// TIA Portal V20 export
// export: Created 2025-12-01T14:56:29.3787725Z, ExportSetting None, DisplayName Totally Integrated Automation Portal, DisplayVersion V20 Update 3, DisplayName TIA Portal Openness, DisplayVersion V20 Update 3, DisplayName TIA Portal Version Control Interface, DisplayVersion V20 Update 3, DisplayName STEP 7 Professional, DisplayVersion V20 Update 3, DisplayName STEP 7 Safety, DisplayVersion V20 Update 2, DisplayName WinCC Basic/Comfort/Advanced, DisplayVersion V20 Update 3, DisplayName WinCC Professional, DisplayVersion V20 Update 3, DisplayName WinCC Unified, DisplayVersion V20 Update 3
FUNCTION_BLOCK "FB430_CRTL_Emp_TP_E1_S23"   // FB430, LAD
{ S7_Optimized_Access := 'FALSE' }
AUTHOR : ROUTER
NAME : 20180827
VERSION : 3.1
// ////////////////////////////////////////////////////////////////
// /  Modificada  24/08/15          NIEVES RODRIGUEZ              /
// /                               /
// ////////////////////////////////////////////////////////////////
// stored: AutoNumber false, SetENOAutomatically false
   VAR_INPUT
      Mesa : UInt;   // Número de mesa
      En_Tension : Bool;
      pHsMx_E1 : Bool;   // pHs de ausencia de la Mesa por E1
      pHsMx_S3 : Bool;   // pHs de ausencia de la Mesa por S3
      Termico_Tx : Bool;   // Proteccion del Tx en E1E3
      Avance_Tx : Bool;   // Avance del Tx
      TP1_Up : Bool;   // TP1 Arriba. E1 >> S3. si no hay tope poner ON
      TP1_Down : Bool;   // TP1 Abajo. E1 >> S3. si no hay tope poner ON
      Simul_Mx : Bool;   // Permiso de Simultaneo en la Entrada E1
      IN_Empuj_recogido : Bool;   // Empujador recogido
      IN_Empuj_Extendido : Bool;   // Empujador extendido
      Mx_Bloq_Activo_S2 : Bool;   // Bloqueo Activo de la Mesa
      AVTF_MAnt_Mx : Bool;   // E1 >> Mesa Anterior AVTF
      PTF_Sal_M3 : Bool;   // S3 >> Mesa Siguiente PTF
      NXT_Avance_S3 : Bool;   // S3 >> Mesa Siguiente avanzando
      PTF_Sal_M2 : Bool;   // Desactiva si Transferencia controlada
      NXT_Avance_S2 : Bool;   // S2 >> Mesa Siguiente avanzando
      F_EnvMens_Mx : Bool;   // Fin de Envio de Mensaje
      Num_Cruce : UInt;   // Número de cruce.
      DB_FIFO_Cruce : UInt := 213;   // DB de la FIFO de ordenes del cruce
      Lng_FIFO_Cruce : UInt := 1;   // Longitut de la FIFO de ordenes del cruce
      ValorOrden_S2 : Word := 16#81;   // Con que orden entra por S2
      MesaS2 : UInt;   // Número de mesa por S2
      MesaS3 : UInt;   // Número de mesa por S3
      V_Paro : UDInt := 4000;   // tiempo que avanza el transportador sin aviso hasta que se para (ms)
      V_CNT_ApHsMx_E1 : UDInt := 500;   // Valor de Ausencia por E1 en ms
      V_CNT_ApHsMx_S3 : UDInt := 500;   // Valor de Ausencia por S3 en ms
      V_Vaciado : UDInt := 3000;   // Valor de vaciado en ms
      V_Gap : UDInt := 200;   // espacio que se deja antes de iniciar un simultaneo en ms
      V_TOut_empujador : UDInt := 2000;   // TimeOut del empujador en ms
      V_TOut_TP : UDInt := 2000;   // TimeOut de Tope en ms
   END_VAR
   VAR_OUTPUT
      P_EnvMens_PMx : Bool;   // Permiso de Enviar Mensaje de Presencia
      Etiqueta_Jdt : UDInt;   // Etiqueta que ha sido leida
      Orden_Ejecutada_Jdt : UInt;   // Orden que se ha ejecutado
      PTF_MAnt_Mx : Bool;   // E1 >> Mesa Anterior PTF
      AVTF_Sal_M3 : Bool;   // S3 >> Mesa Siguiente AVTF
      NXT_Descarga_Act_S3 : Bool;   // S3 >> Mesa Siguiente Descarga activa
      AVTF_Sal_M2 : Bool;   // S2 >> Mesa Siguiente AVTF
      NXT_Descarga_Act_S2 : Bool;   // S2 >> Mesa Siguiente Descarga activa
   END_VAR
   VAR
      T1_ET00 : Bool;
      T1_ET01 : Bool;
      T1_ET02 : Bool;
      T1_ET03 : Bool;
      T1_ET10 : Bool;
      T1_ET11 : Bool;
      T1_ET50 : Bool;
      T1_ET60 : Bool;
      T1_ET61 : Bool;
      T1_ET110 : Bool;
      T1_ET111 : Bool;
      T1_ET112 : Bool;
      FIFO_OK : Bool;
      TRANS_OK : Bool;
      O_Bloqueo : Bool;
      FN_ET02 : Bool;
      FP_ET50 : Bool;
      FP_Bajar_TP : Bool;
      TOUT_empujador : Bool;
      ok_vaciado : Bool;
      maux_fp_disparo : Bool;
      maux_fn_s3 : Bool;
      maux_fn_e1 : Bool;
      mem_fn_e1 : Bool;
      mem_fn_s3 : Bool;
      TmpSIMUL : UDInt;
      Tmp_Ausencia : UDInt;
      Tmp_Vaciado : UDInt;
      tmp_tout_empujador : UDInt;
      Tmp_tout_tope : UDInt;
      tmp_ausencia_S3 : UDInt;
      TMP_Paro : UDInt;
      TMP_En_tension : UDInt;
      Datos_Scanner { S7_SetPoint := 'True'} : "ROUT_Orden_Fifo_Scanner";
   END_VAR
   VAR_TEMP
      EstadoZona : "EstadoZona";   // Estado de Zona de la Mesa
      EstadoVI : "EstadosMesa";   // Estado del Vehiculo Inteliguente de la Mesa
      ConfigFB : "UDT_ConfigFB";   // Configuracion de la FB de la Mesa
      OK_tension : Bool;
      MA_SubirTP : Bool;
      O_Sal_S3 : Bool;
      O_Sal_S2 : Bool;
      O_Vaciar : Bool;
      Moti_ERRO : Bool;
      Moti_NENC : Bool;
      Moti_NORM : Bool;
      Moti_INIC : Bool;
      OK_SIMUL_S3 : Bool;
      ok_ausencia_S3 : Bool;
      tout_tope : Bool;
      ok_ausencia_E1 : Bool;
      tiempo_paro_ok : Bool;
      INT_ORDEN : UInt;
      I_Ord_Filtrada : UInt;
      I_V_Ord_Entrar : UInt;
      Prox_Orden : UInt;
      Prox_Etiqueta : DInt;
      Aux_W_Orden : Word;
      Aux_W_Moti : Word;
   END_VAR
   VAR_TEMP   // added for the SCL form of the ladder/FBD networks
      _w1 : Bool;
      _w2 : Bool;
      _w3 : Bool;
      _w4 : Bool;
      _w5 : Bool;
      _w6 : Bool;
   END_VAR
BEGIN

REGION Network 1: INICIALIZAR - Recoger las Variables de Estado de la Mesa
   // Se recoge - Estado_CBx
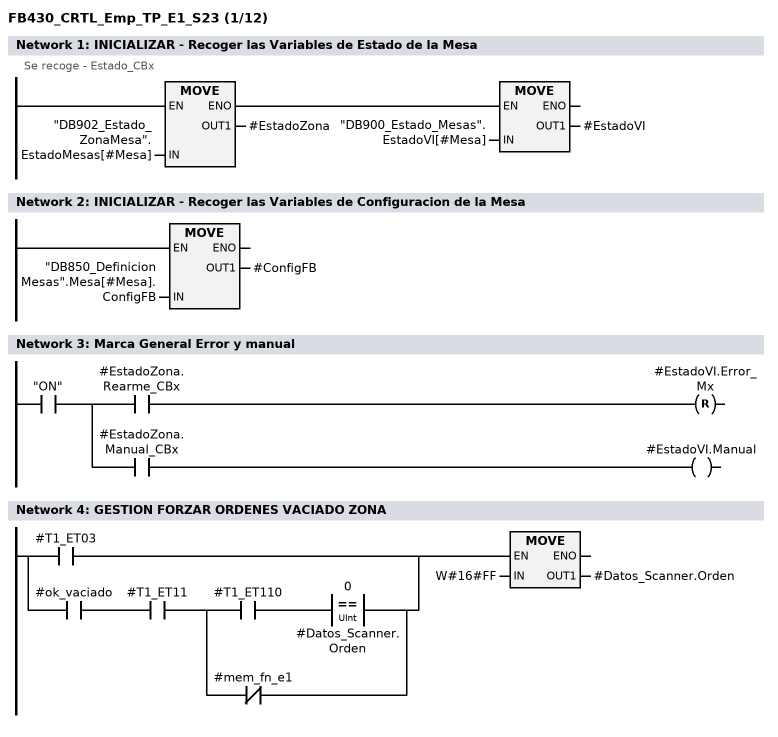
   RUNG wire#powerrail
      Move(in := "DB902_Estado_ZonaMesa".EstadoMesas[#Mesa], out1 => #EstadoZona)
      Move(in := "DB900_Estado_Mesas".EstadoVI[#Mesa], out1 => #EstadoVI)
   END_RUNG
   // the same network as SCL:
   #EstadoZona := "DB902_Estado_ZonaMesa".EstadoMesas[#Mesa];
   #EstadoVI := "DB900_Estado_Mesas".EstadoVI[#Mesa];
END_REGION

REGION Network 2: INICIALIZAR - Recoger las Variables de Configuracion de la Mesa
   RUNG wire#powerrail
      Move(in := "DB850_DefinicionMesas".Mesa[#Mesa].ConfigFB, out1 => #ConfigFB)
   END_RUNG
   // the same network as SCL:
   #ConfigFB := "DB850_DefinicionMesas".Mesa[#Mesa].ConfigFB;
END_REGION

REGION Network 3: Marca General Error y manual
   RUNG wire#powerrail
      Contact( "ON" )
      wire#w1
      Contact( #EstadoZona.Rearme_CBx )
      R_Coil( #EstadoVI.Error_Mx )
   END_RUNG
   RUNG wire#w1
      Contact( #EstadoZona.Manual_CBx )
      Coil( #EstadoVI.Manual )
   END_RUNG
   // the same network as SCL:
   IF "ON" AND #EstadoZona.Rearme_CBx THEN #EstadoVI.Error_Mx := FALSE; END_IF;
   #EstadoVI.Manual := "ON" AND #EstadoZona.Manual_CBx;
END_REGION

REGION Network 4: GESTION FORZAR ORDENES VACIADO ZONA
   RUNG wire#powerrail
      Contact( #T1_ET03 )
      wire#w1
      { S7_GenerateENO := "TRUE" } Move(in := W#16#FF, out1 => #Datos_Scanner.Orden)
   END_RUNG
   RUNG wire#powerrail
      Contact( #ok_vaciado )
      Contact( #T1_ET11 )
      wire#w2
      Contact( #T1_ET110 )
      { S7_Templates := "SrcType := UInt" } EQ_Contact(in1 := 0, in2 := #Datos_Scanner.Orden)
   END_RUNG wire#w1
   RUNG wire#w2
      I_Contact( #mem_fn_e1 )
   END_RUNG wire#w1
   // the same network as SCL:
   IF #T1_ET03 OR (#ok_vaciado AND #T1_ET11 AND ((#T1_ET110 AND (0 = #Datos_Scanner.Orden)) OR NOT #mem_fn_e1)) THEN
       #Datos_Scanner.Orden := W#16#FF;
   END_IF;
END_REGION

REGION Network 5: Extraccion de orden
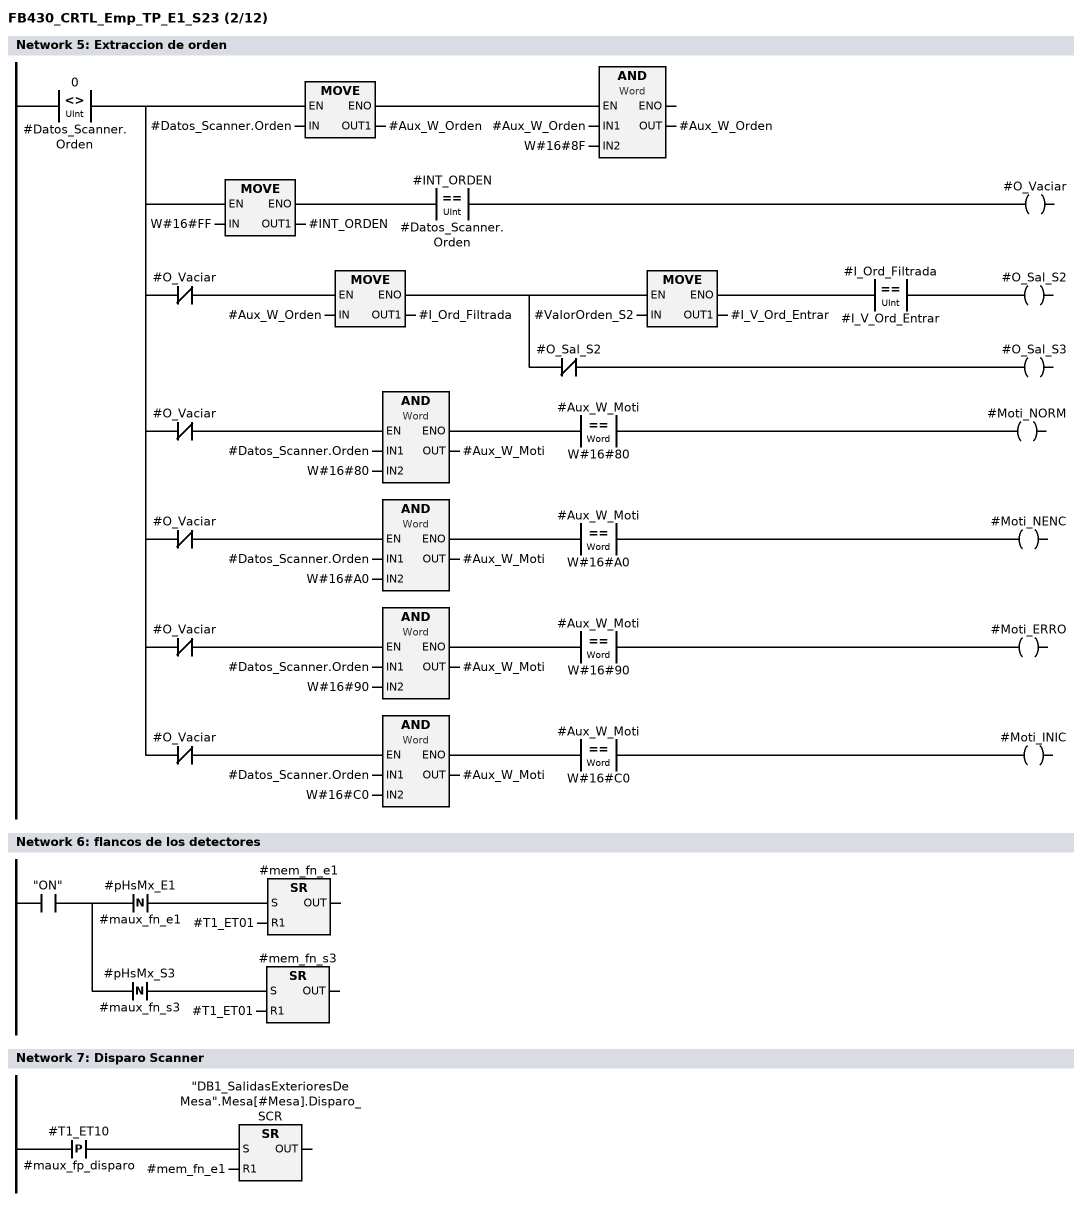
   RUNG wire#powerrail
      { S7_Templates := "SrcType := UInt" } NE_Contact(in1 := 0, in2 := #Datos_Scanner.Orden)
      wire#w1
      { S7_GenerateENO := "TRUE" } Move(in := #Datos_Scanner.Orden, out1 => #Aux_W_Orden)
      { S7_Templates := "SrcType := Word"; S7_GenerateENO := "TRUE" } And(in1 := #Aux_W_Orden, in2 := W#16#8F, out => #Aux_W_Orden)
   END_RUNG
   RUNG wire#w1
      { S7_GenerateENO := "TRUE" } Move(in := W#16#FF, out1 => #INT_ORDEN)
      { S7_Templates := "SrcType := UInt" } EQ_Contact(in1 := #INT_ORDEN, in2 := #Datos_Scanner.Orden)
      Coil( #O_Vaciar )
   END_RUNG
   RUNG wire#w1
      I_Contact( #O_Vaciar )
      { S7_GenerateENO := "TRUE" } Move(in := #Aux_W_Orden, out1 => #I_Ord_Filtrada)
      wire#w2
      { S7_GenerateENO := "TRUE" } Move(in := #ValorOrden_S2, out1 => #I_V_Ord_Entrar)
      { S7_Templates := "SrcType := UInt" } EQ_Contact(in1 := #I_Ord_Filtrada, in2 := #I_V_Ord_Entrar)
      Coil( #O_Sal_S2 )
   END_RUNG
   RUNG wire#w2
      I_Contact( #O_Sal_S2 )
      Coil( #O_Sal_S3 )
   END_RUNG
   RUNG wire#w1
      I_Contact( #O_Vaciar )
      { S7_Templates := "SrcType := Word"; S7_GenerateENO := "TRUE" } And(in1 := #Datos_Scanner.Orden, in2 := W#16#80, out => #Aux_W_Moti)
      { S7_Templates := "SrcType := Word" } EQ_Contact(in1 := #Aux_W_Moti, in2 := W#16#80)
      Coil( #Moti_NORM )
   END_RUNG
   RUNG wire#w1
      I_Contact( #O_Vaciar )
      { S7_Templates := "SrcType := Word"; S7_GenerateENO := "TRUE" } And(in1 := #Datos_Scanner.Orden, in2 := W#16#A0, out => #Aux_W_Moti)
      { S7_Templates := "SrcType := Word" } EQ_Contact(in1 := #Aux_W_Moti, in2 := W#16#A0)
      Coil( #Moti_NENC )
   END_RUNG
   RUNG wire#w1
      I_Contact( #O_Vaciar )
      { S7_Templates := "SrcType := Word"; S7_GenerateENO := "TRUE" } And(in1 := #Datos_Scanner.Orden, in2 := W#16#90, out => #Aux_W_Moti)
      { S7_Templates := "SrcType := Word" } EQ_Contact(in1 := #Aux_W_Moti, in2 := W#16#90)
      Coil( #Moti_ERRO )
   END_RUNG
   RUNG wire#w1
      I_Contact( #O_Vaciar )
      { S7_Templates := "SrcType := Word"; S7_GenerateENO := "TRUE" } And(in1 := #Datos_Scanner.Orden, in2 := W#16#C0, out => #Aux_W_Moti)
      { S7_Templates := "SrcType := Word" } EQ_Contact(in1 := #Aux_W_Moti, in2 := W#16#C0)
      Coil( #Moti_INIC )
   END_RUNG
   // the same network as SCL:
   // ENO of a box is taken as its EN; it also drops when the box reports an error
   #_w1 := 0 <> #Datos_Scanner.Orden;
   IF #_w1 THEN
       #Aux_W_Orden := #Datos_Scanner.Orden;
       #Aux_W_Orden := #Aux_W_Orden AND W#16#8F;
       #INT_ORDEN := W#16#FF;
   END_IF;
   #O_Vaciar := #_w1 AND (#INT_ORDEN = #Datos_Scanner.Orden);
   #_w2 := #_w1 AND NOT #O_Vaciar;
   IF #_w2 THEN
       #I_Ord_Filtrada := #Aux_W_Orden;
       #I_V_Ord_Entrar := #ValorOrden_S2;
   END_IF;
   #O_Sal_S2 := #_w2 AND (#I_Ord_Filtrada = #I_V_Ord_Entrar);
   #O_Sal_S3 := #_w2 AND NOT #O_Sal_S2;
   #_w3 := #_w1 AND NOT #O_Vaciar;
   IF #_w3 THEN #Aux_W_Moti := #Datos_Scanner.Orden AND W#16#80; END_IF;
   #Moti_NORM := #_w3 AND (#Aux_W_Moti = W#16#80);
   #_w4 := #_w1 AND NOT #O_Vaciar;
   IF #_w4 THEN #Aux_W_Moti := #Datos_Scanner.Orden AND W#16#A0; END_IF;
   #Moti_NENC := #_w4 AND (#Aux_W_Moti = W#16#A0);
   #_w5 := #_w1 AND NOT #O_Vaciar;
   IF #_w5 THEN #Aux_W_Moti := #Datos_Scanner.Orden AND W#16#90; END_IF;
   #Moti_ERRO := #_w5 AND (#Aux_W_Moti = W#16#90);
   #_w6 := #_w1 AND NOT #O_Vaciar;
   IF #_w6 THEN #Aux_W_Moti := #Datos_Scanner.Orden AND W#16#C0; END_IF;
   #Moti_INIC := #_w6 AND (#Aux_W_Moti = W#16#C0);
END_REGION

REGION Network 6: flancos de los detectores
   RUNG wire#powerrail
      Contact( "ON" )
      wire#w1
      N_Contact(operand := #pHsMx_E1, bit := #maux_fn_e1)
      S_SR(operand := #mem_fn_e1, r1 := #T1_ET01)
   END_RUNG
   RUNG wire#w1
      N_Contact(operand := #pHsMx_S3, bit := #maux_fn_s3)
      S_SR(operand := #mem_fn_s3, r1 := #T1_ET01)
   END_RUNG
   // the same network as SCL:
   #_w1 := "ON" AND NOT #pHsMx_E1 AND #maux_fn_e1;   // falling edge of #pHsMx_E1
   #maux_fn_e1 := #pHsMx_E1;
   IF #_w1 THEN
       #mem_fn_e1 := TRUE;   // SR flip-flop
   END_IF;
   IF #T1_ET01 THEN #mem_fn_e1 := FALSE; END_IF;
   #_w2 := "ON" AND NOT #pHsMx_S3 AND #maux_fn_s3;   // falling edge of #pHsMx_S3
   #maux_fn_s3 := #pHsMx_S3;
   IF #_w2 THEN
       #mem_fn_s3 := TRUE;   // SR flip-flop
   END_IF;
   IF #T1_ET01 THEN #mem_fn_s3 := FALSE; END_IF;
END_REGION

REGION Network 7: Disparo Scanner
   RUNG wire#powerrail
      P_Contact(operand := #T1_ET10, bit := #maux_fp_disparo)
      S_SR(operand := "DB1_SalidasExterioresDeMesa".Mesa[#Mesa].Disparo_SCR, r1 := #mem_fn_e1)
   END_RUNG
   // the same network as SCL:
   #_w1 := #T1_ET10 AND NOT #maux_fp_disparo;   // rising edge of #T1_ET10
   #maux_fp_disparo := #T1_ET10;
   IF #_w1 THEN
       "DB1_SalidasExterioresDeMesa".Mesa[#Mesa].Disparo_SCR := TRUE;   // SR flip-flop
   END_IF;
   IF #mem_fn_e1 THEN "DB1_SalidasExterioresDeMesa".Mesa[#Mesa].Disparo_SCR := FALSE; END_IF;
END_REGION

REGION Network 8: Contador de ausencia E1
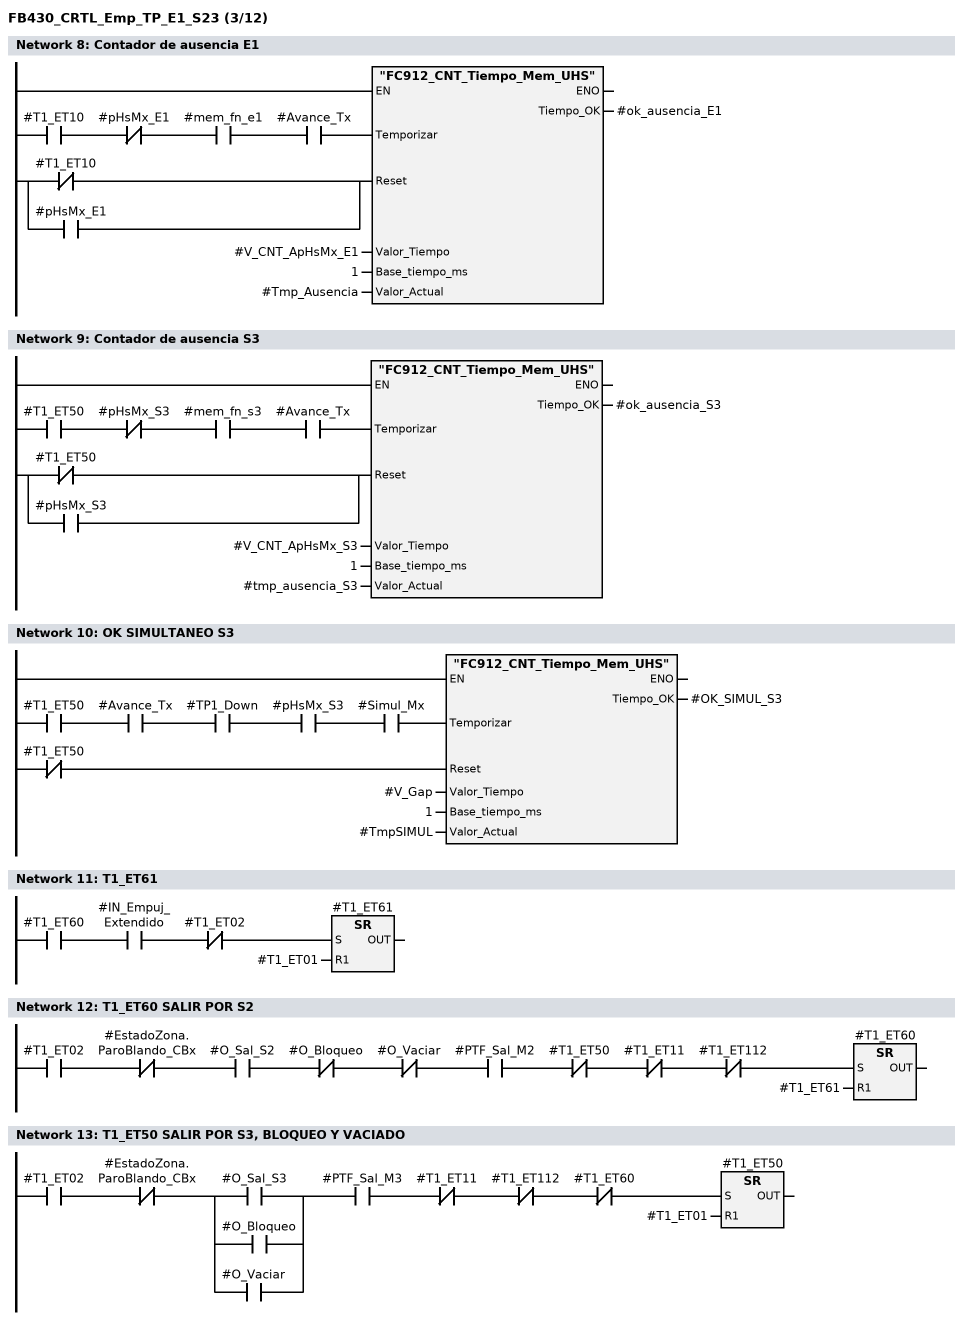
   RUNG wire#powerrail
      "FC912_CNT_Tiempo_Mem_UHS"(Temporizar := wire#w1, Reset := wire#w2, Valor_Tiempo := #V_CNT_ApHsMx_E1, Base_tiempo_ms := 1, Valor_Actual := #Tmp_Ausencia, Tiempo_OK => #ok_ausencia_E1)
   END_RUNG
   RUNG wire#powerrail
      Contact( #T1_ET10 )
      I_Contact( #pHsMx_E1 )
      Contact( #mem_fn_e1 )
      Contact( #Avance_Tx )
   END_RUNG wire#w1
   RUNG wire#powerrail
      I_Contact( #T1_ET10 )
   END_RUNG wire#w2
   RUNG wire#powerrail
      Contact( #pHsMx_E1 )
   END_RUNG wire#w2
   // the same network as SCL:
   "FC912_CNT_Tiempo_Mem_UHS"(Temporizar := #T1_ET10 AND NOT #pHsMx_E1 AND #mem_fn_e1 AND #Avance_Tx,
                           Reset := NOT #T1_ET10 OR #pHsMx_E1,
                           Valor_Tiempo := #V_CNT_ApHsMx_E1,
                           Base_tiempo_ms := 1,
                           Valor_Actual := #Tmp_Ausencia,
                           Tiempo_OK => #ok_ausencia_E1);
END_REGION

REGION Network 9: Contador de ausencia S3
   RUNG wire#powerrail
      "FC912_CNT_Tiempo_Mem_UHS"(Temporizar := wire#w1, Reset := wire#w2, Valor_Tiempo := #V_CNT_ApHsMx_S3, Base_tiempo_ms := 1, Valor_Actual := #tmp_ausencia_S3, Tiempo_OK => #ok_ausencia_S3)
   END_RUNG
   RUNG wire#powerrail
      Contact( #T1_ET50 )
      I_Contact( #pHsMx_S3 )
      Contact( #mem_fn_s3 )
      Contact( #Avance_Tx )
   END_RUNG wire#w1
   RUNG wire#powerrail
      I_Contact( #T1_ET50 )
   END_RUNG wire#w2
   RUNG wire#powerrail
      Contact( #pHsMx_S3 )
   END_RUNG wire#w2
   // the same network as SCL:
   "FC912_CNT_Tiempo_Mem_UHS"(Temporizar := #T1_ET50 AND NOT #pHsMx_S3 AND #mem_fn_s3 AND #Avance_Tx,
                           Reset := NOT #T1_ET50 OR #pHsMx_S3,
                           Valor_Tiempo := #V_CNT_ApHsMx_S3,
                           Base_tiempo_ms := 1,
                           Valor_Actual := #tmp_ausencia_S3,
                           Tiempo_OK => #ok_ausencia_S3);
END_REGION

REGION Network 10: OK SIMULTANEO S3
   RUNG wire#powerrail
      "FC912_CNT_Tiempo_Mem_UHS"(Temporizar := wire#w1, Reset := wire#w2, Valor_Tiempo := #V_Gap, Base_tiempo_ms := 1, Valor_Actual := #TmpSIMUL, Tiempo_OK => #OK_SIMUL_S3)
   END_RUNG
   RUNG wire#powerrail
      Contact( #T1_ET50 )
      Contact( #Avance_Tx )
      Contact( #TP1_Down )
      Contact( #pHsMx_S3 )
      Contact( #Simul_Mx )
   END_RUNG wire#w1
   RUNG wire#powerrail
      I_Contact( #T1_ET50 )
   END_RUNG wire#w2
   // the same network as SCL:
   "FC912_CNT_Tiempo_Mem_UHS"(Temporizar := #T1_ET50 AND #Avance_Tx AND #TP1_Down AND #pHsMx_S3 AND #Simul_Mx,
                           Reset := NOT #T1_ET50,
                           Valor_Tiempo := #V_Gap,
                           Base_tiempo_ms := 1,
                           Valor_Actual := #TmpSIMUL,
                           Tiempo_OK => #OK_SIMUL_S3);
END_REGION

REGION Network 11: T1_ET61
   RUNG wire#powerrail
      Contact( #T1_ET60 )
      Contact( #IN_Empuj_Extendido )
      I_Contact( #T1_ET02 )
      S_SR(operand := #T1_ET61, r1 := #T1_ET01)
   END_RUNG
   // the same network as SCL:
   IF #T1_ET60 AND #IN_Empuj_Extendido AND NOT #T1_ET02 THEN
       #T1_ET61 := TRUE;   // SR flip-flop
   END_IF;
   IF #T1_ET01 THEN #T1_ET61 := FALSE; END_IF;
END_REGION

REGION Network 12: T1_ET60 SALIR POR S2
   RUNG wire#powerrail
      Contact( #T1_ET02 )
      I_Contact( #EstadoZona.ParoBlando_CBx )
      Contact( #O_Sal_S2 )
      I_Contact( #O_Bloqueo )
      I_Contact( #O_Vaciar )
      Contact( #PTF_Sal_M2 )
      I_Contact( #T1_ET50 )
      I_Contact( #T1_ET11 )
      I_Contact( #T1_ET112 )
      S_SR(operand := #T1_ET60, r1 := #T1_ET61)
   END_RUNG
   // the same network as SCL:
   IF #T1_ET02 AND NOT #EstadoZona.ParoBlando_CBx AND #O_Sal_S2 AND NOT #O_Bloqueo AND NOT #O_Vaciar AND #PTF_Sal_M2 AND NOT #T1_ET50 AND NOT #T1_ET11 AND NOT #T1_ET112 THEN
       #T1_ET60 := TRUE;   // SR flip-flop
   END_IF;
   IF #T1_ET61 THEN #T1_ET60 := FALSE; END_IF;
END_REGION

REGION Network 13: T1_ET50 SALIR POR S3, BLOQUEO Y VACIADO
   RUNG wire#powerrail
      Contact( #T1_ET02 )
      I_Contact( #EstadoZona.ParoBlando_CBx )
      wire#w1
      Contact( #O_Sal_S3 )
      wire#w2
      Contact( #PTF_Sal_M3 )
      I_Contact( #T1_ET11 )
      I_Contact( #T1_ET112 )
      I_Contact( #T1_ET60 )
      S_SR(operand := #T1_ET50, r1 := #T1_ET01)
   END_RUNG
   RUNG wire#w1
      Contact( #O_Bloqueo )
   END_RUNG wire#w2
   RUNG wire#w1
      Contact( #O_Vaciar )
   END_RUNG wire#w2
   // the same network as SCL:
   IF #T1_ET02 AND NOT #EstadoZona.ParoBlando_CBx AND (#O_Sal_S3 OR #O_Bloqueo OR #O_Vaciar) AND #PTF_Sal_M3 AND NOT #T1_ET11 AND NOT #T1_ET112 AND NOT #T1_ET60 THEN
       #T1_ET50 := TRUE;   // SR flip-flop
   END_IF;
   IF #T1_ET01 THEN #T1_ET50 := FALSE; END_IF;
END_REGION

REGION Network 14: T1_ET02 ESTADO REPOSO CARGADA
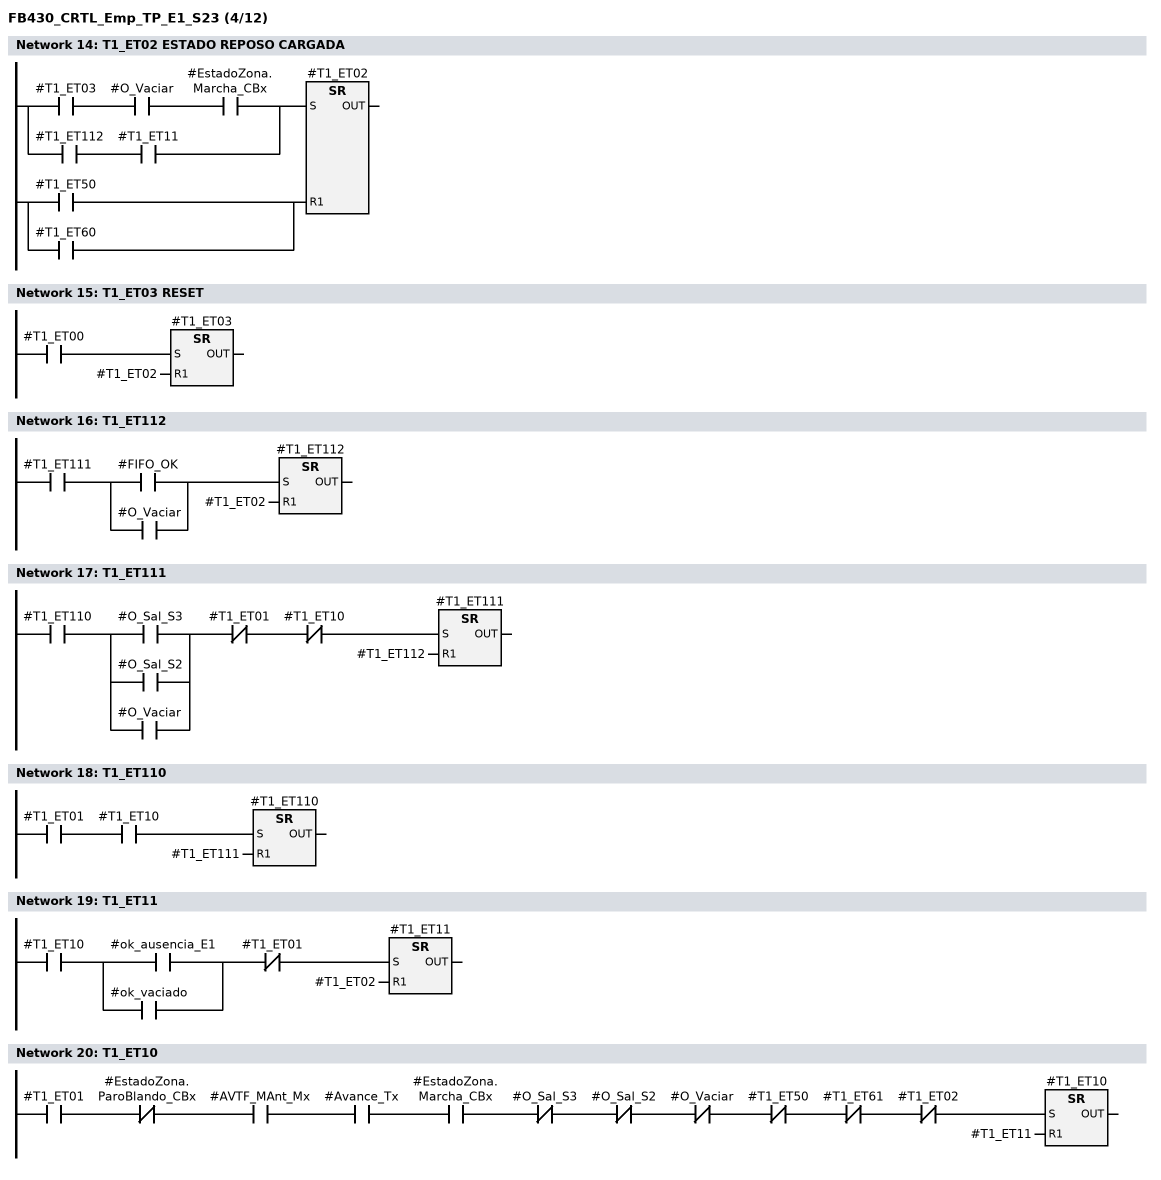
   RUNG wire#powerrail
      Contact( #T1_ET03 )
      Contact( #O_Vaciar )
      Contact( #EstadoZona.Marcha_CBx )
      wire#w1
      S_SR(operand := #T1_ET02, r1 := wire#w2)
   END_RUNG
   RUNG wire#powerrail
      Contact( #T1_ET112 )
      Contact( #T1_ET11 )
   END_RUNG wire#w1
   RUNG wire#powerrail
      Contact( #T1_ET50 )
   END_RUNG wire#w2
   RUNG wire#powerrail
      Contact( #T1_ET60 )
   END_RUNG wire#w2
   // the same network as SCL:
   IF (#T1_ET03 AND #O_Vaciar AND #EstadoZona.Marcha_CBx) OR (#T1_ET112 AND #T1_ET11) THEN
       #T1_ET02 := TRUE;   // SR flip-flop
   END_IF;
   IF #T1_ET50 OR #T1_ET60 THEN #T1_ET02 := FALSE; END_IF;
END_REGION

REGION Network 15: T1_ET03 RESET
   RUNG wire#powerrail
      Contact( #T1_ET00 )
      S_SR(operand := #T1_ET03, r1 := #T1_ET02)
   END_RUNG
   // the same network as SCL:
   IF #T1_ET00 THEN
       #T1_ET03 := TRUE;   // SR flip-flop
   END_IF;
   IF #T1_ET02 THEN #T1_ET03 := FALSE; END_IF;
END_REGION

REGION Network 16: T1_ET112
   RUNG wire#powerrail
      Contact( #T1_ET111 )
      wire#w1
      Contact( #FIFO_OK )
      wire#w2
      S_SR(operand := #T1_ET112, r1 := #T1_ET02)
   END_RUNG
   RUNG wire#w1
      Contact( #O_Vaciar )
   END_RUNG wire#w2
   // the same network as SCL:
   IF #T1_ET111 AND (#FIFO_OK OR #O_Vaciar) THEN
       #T1_ET112 := TRUE;   // SR flip-flop
   END_IF;
   IF #T1_ET02 THEN #T1_ET112 := FALSE; END_IF;
END_REGION

REGION Network 17: T1_ET111
   RUNG wire#powerrail
      Contact( #T1_ET110 )
      wire#w1
      Contact( #O_Sal_S3 )
      wire#w2
      I_Contact( #T1_ET01 )
      I_Contact( #T1_ET10 )
      S_SR(operand := #T1_ET111, r1 := #T1_ET112)
   END_RUNG
   RUNG wire#w1
      Contact( #O_Sal_S2 )
   END_RUNG wire#w2
   RUNG wire#w1
      Contact( #O_Vaciar )
   END_RUNG wire#w2
   // the same network as SCL:
   IF #T1_ET110 AND (#O_Sal_S3 OR #O_Sal_S2 OR #O_Vaciar) AND NOT #T1_ET01 AND NOT #T1_ET10 THEN
       #T1_ET111 := TRUE;   // SR flip-flop
   END_IF;
   IF #T1_ET112 THEN #T1_ET111 := FALSE; END_IF;
END_REGION

REGION Network 18: T1_ET110
   RUNG wire#powerrail
      Contact( #T1_ET01 )
      Contact( #T1_ET10 )
      S_SR(operand := #T1_ET110, r1 := #T1_ET111)
   END_RUNG
   // the same network as SCL:
   IF #T1_ET01 AND #T1_ET10 THEN
       #T1_ET110 := TRUE;   // SR flip-flop
   END_IF;
   IF #T1_ET111 THEN #T1_ET110 := FALSE; END_IF;
END_REGION

REGION Network 19: T1_ET11
   RUNG wire#powerrail
      Contact( #T1_ET10 )
      wire#w1
      Contact( #ok_ausencia_E1 )
      wire#w2
      I_Contact( #T1_ET01 )
      S_SR(operand := #T1_ET11, r1 := #T1_ET02)
   END_RUNG
   RUNG wire#w1
      Contact( #ok_vaciado )
   END_RUNG wire#w2
   // the same network as SCL:
   IF #T1_ET10 AND (#ok_ausencia_E1 OR #ok_vaciado) AND NOT #T1_ET01 THEN
       #T1_ET11 := TRUE;   // SR flip-flop
   END_IF;
   IF #T1_ET02 THEN #T1_ET11 := FALSE; END_IF;
END_REGION

REGION Network 20: T1_ET10
   RUNG wire#powerrail
      Contact( #T1_ET01 )
      I_Contact( #EstadoZona.ParoBlando_CBx )
      Contact( #AVTF_MAnt_Mx )
      Contact( #Avance_Tx )
      Contact( #EstadoZona.Marcha_CBx )
      I_Contact( #O_Sal_S3 )
      I_Contact( #O_Sal_S2 )
      I_Contact( #O_Vaciar )
      I_Contact( #T1_ET50 )
      I_Contact( #T1_ET61 )
      I_Contact( #T1_ET02 )
      S_SR(operand := #T1_ET10, r1 := #T1_ET11)
   END_RUNG
   // the same network as SCL:
   IF #T1_ET01 AND NOT #EstadoZona.ParoBlando_CBx AND #AVTF_MAnt_Mx AND #Avance_Tx AND #EstadoZona.Marcha_CBx AND NOT #O_Sal_S3 AND NOT #O_Sal_S2 AND NOT #O_Vaciar AND NOT #T1_ET50 AND NOT #T1_ET61 AND NOT #T1_ET02 THEN
       #T1_ET10 := TRUE;   // SR flip-flop
   END_IF;
   IF #T1_ET11 THEN #T1_ET10 := FALSE; END_IF;
END_REGION

REGION Network 21: T1_ET01 ESTADO REPOSO VACIO
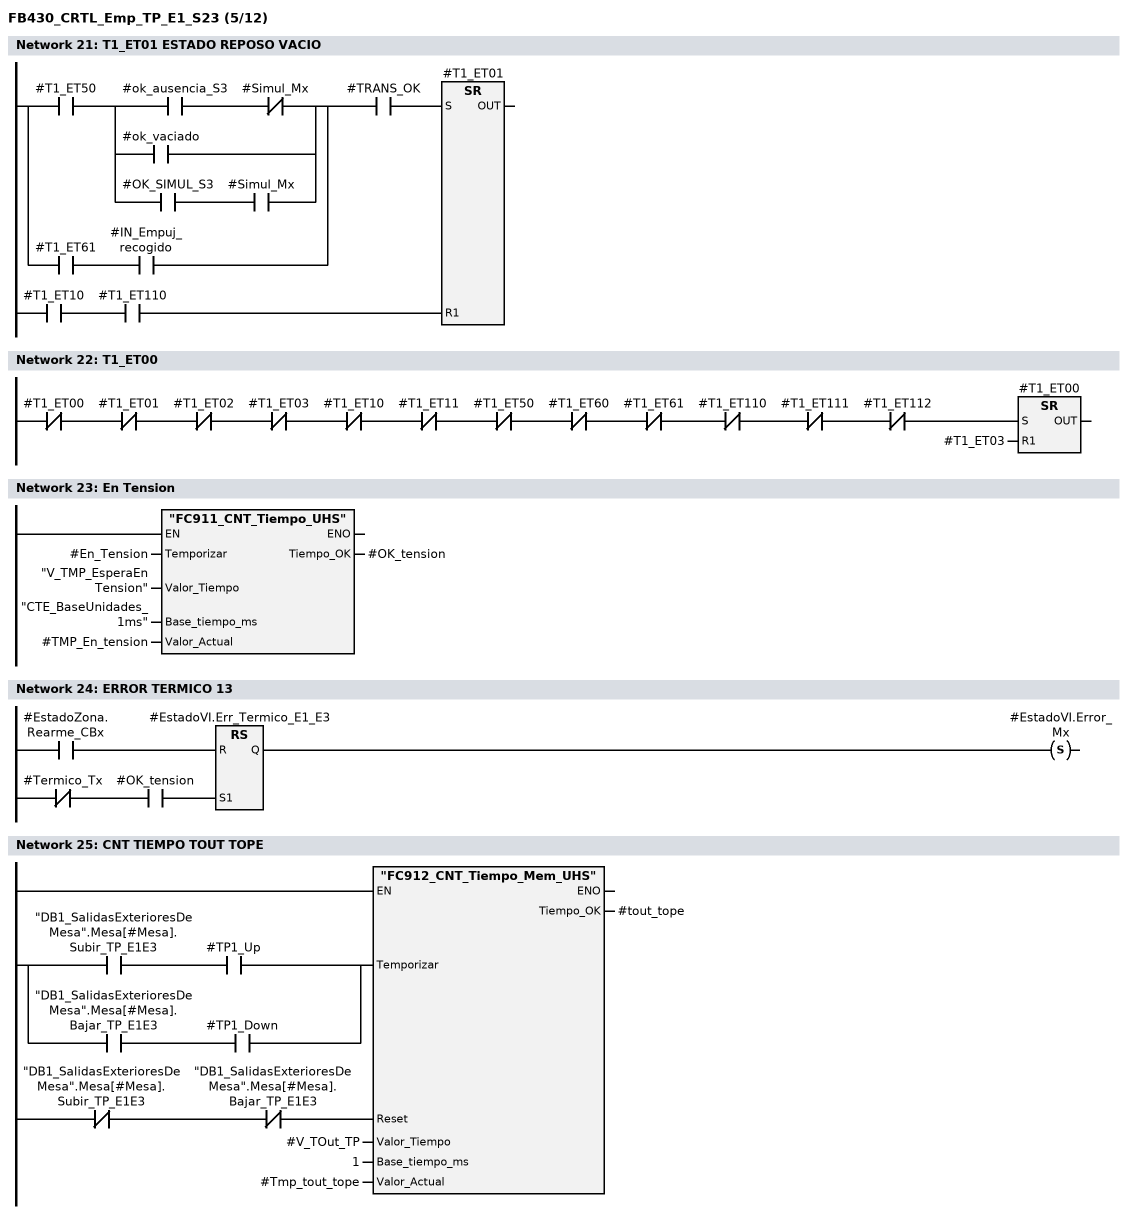
   RUNG wire#powerrail
      Contact( #T1_ET50 )
      wire#w1
      Contact( #ok_ausencia_S3 )
      I_Contact( #Simul_Mx )
      wire#w2
      Contact( #TRANS_OK )
      S_SR(operand := #T1_ET01, r1 := wire#w3)
   END_RUNG
   RUNG wire#w1
      Contact( #ok_vaciado )
   END_RUNG wire#w2
   RUNG wire#w1
      Contact( #OK_SIMUL_S3 )
      Contact( #Simul_Mx )
   END_RUNG wire#w2
   RUNG wire#powerrail
      Contact( #T1_ET61 )
      Contact( #IN_Empuj_recogido )
   END_RUNG wire#w2
   RUNG wire#powerrail
      Contact( #T1_ET10 )
      Contact( #T1_ET110 )
   END_RUNG wire#w3
   // the same network as SCL:
   IF ((#T1_ET50 AND ((#ok_ausencia_S3 AND NOT #Simul_Mx) OR #ok_vaciado OR (#OK_SIMUL_S3 AND #Simul_Mx))) OR (#T1_ET61 AND #IN_Empuj_recogido)) AND #TRANS_OK THEN
       #T1_ET01 := TRUE;   // SR flip-flop
   END_IF;
   IF #T1_ET10 AND #T1_ET110 THEN #T1_ET01 := FALSE; END_IF;
END_REGION

REGION Network 22: T1_ET00
   RUNG wire#powerrail
      I_Contact( #T1_ET00 )
      I_Contact( #T1_ET01 )
      I_Contact( #T1_ET02 )
      I_Contact( #T1_ET03 )
      I_Contact( #T1_ET10 )
      I_Contact( #T1_ET11 )
      I_Contact( #T1_ET50 )
      I_Contact( #T1_ET60 )
      I_Contact( #T1_ET61 )
      I_Contact( #T1_ET110 )
      I_Contact( #T1_ET111 )
      I_Contact( #T1_ET112 )
      S_SR(operand := #T1_ET00, r1 := #T1_ET03)
   END_RUNG
   // the same network as SCL:
   IF NOT #T1_ET00 AND NOT #T1_ET01 AND NOT #T1_ET02 AND NOT #T1_ET03 AND NOT #T1_ET10 AND NOT #T1_ET11 AND NOT #T1_ET50 AND NOT #T1_ET60 AND NOT #T1_ET61 AND NOT #T1_ET110 AND NOT #T1_ET111 AND NOT #T1_ET112 THEN
       #T1_ET00 := TRUE;   // SR flip-flop
   END_IF;
   IF #T1_ET03 THEN #T1_ET00 := FALSE; END_IF;
END_REGION

REGION Network 23: En Tension
   RUNG wire#powerrail
      "FC911_CNT_Tiempo_UHS"(Temporizar := #En_Tension, Valor_Tiempo := "V_TMP_EsperaEnTension", Base_tiempo_ms := "CTE_BaseUnidades_1ms", Valor_Actual := #TMP_En_tension, Tiempo_OK => #OK_tension)
   END_RUNG
   // the same network as SCL:
   "FC911_CNT_Tiempo_UHS"(Temporizar := #En_Tension,
                          Valor_Tiempo := "V_TMP_EsperaEnTension",
                          Base_tiempo_ms := "CTE_BaseUnidades_1ms",
                          Valor_Actual := #TMP_En_tension,
                          Tiempo_OK => #OK_tension);
END_REGION

REGION Network 24: ERROR TERMICO 13
   RUNG wire#powerrail
      Contact( #EstadoZona.Rearme_CBx )
      S_RS(operand := #EstadoVI.Err_Termico_E1_E3, s1 := wire#w1)
      S_Coil( #EstadoVI.Error_Mx )
   END_RUNG
   RUNG wire#powerrail
      I_Contact( #Termico_Tx )
      Contact( #OK_tension )
   END_RUNG wire#w1
   // the same network as SCL:
   IF #EstadoZona.Rearme_CBx THEN
       #EstadoVI.Err_Termico_E1_E3 := FALSE;   // RS flip-flop
   END_IF;
   IF NOT #Termico_Tx AND #OK_tension THEN #EstadoVI.Err_Termico_E1_E3 := TRUE; END_IF;
   IF #EstadoVI.Err_Termico_E1_E3 THEN #EstadoVI.Error_Mx := TRUE; END_IF;
END_REGION

REGION Network 25: CNT TIEMPO TOUT TOPE
   RUNG wire#powerrail
      "FC912_CNT_Tiempo_Mem_UHS"(Temporizar := wire#w1, Reset := wire#w2, Valor_Tiempo := #V_TOut_TP, Base_tiempo_ms := 1, Valor_Actual := #Tmp_tout_tope, Tiempo_OK => #tout_tope)
   END_RUNG
   RUNG wire#powerrail
      Contact( "DB1_SalidasExterioresDeMesa".Mesa[#Mesa].Subir_TP_E1E3 )
      Contact( #TP1_Up )
   END_RUNG wire#w1
   RUNG wire#powerrail
      Contact( "DB1_SalidasExterioresDeMesa".Mesa[#Mesa].Bajar_TP_E1E3 )
      Contact( #TP1_Down )
   END_RUNG wire#w1
   RUNG wire#powerrail
      I_Contact( "DB1_SalidasExterioresDeMesa".Mesa[#Mesa].Subir_TP_E1E3 )
      I_Contact( "DB1_SalidasExterioresDeMesa".Mesa[#Mesa].Bajar_TP_E1E3 )
   END_RUNG wire#w2
   // the same network as SCL:
   "FC912_CNT_Tiempo_Mem_UHS"(Temporizar := ("DB1_SalidasExterioresDeMesa".Mesa[#Mesa].Subir_TP_E1E3 AND #TP1_Up) OR ("DB1_SalidasExterioresDeMesa".Mesa[#Mesa].Bajar_TP_E1E3 AND #TP1_Down),
                           Reset := NOT "DB1_SalidasExterioresDeMesa".Mesa[#Mesa].Subir_TP_E1E3 AND NOT "DB1_SalidasExterioresDeMesa".Mesa[#Mesa].Bajar_TP_E1E3,
                           Valor_Tiempo := #V_TOut_TP,
                           Base_tiempo_ms := 1,
                           Valor_Actual := #Tmp_tout_tope,
                           Tiempo_OK => #tout_tope);
END_REGION

REGION Network 26: ERROR TOUT TOPE SUBIR
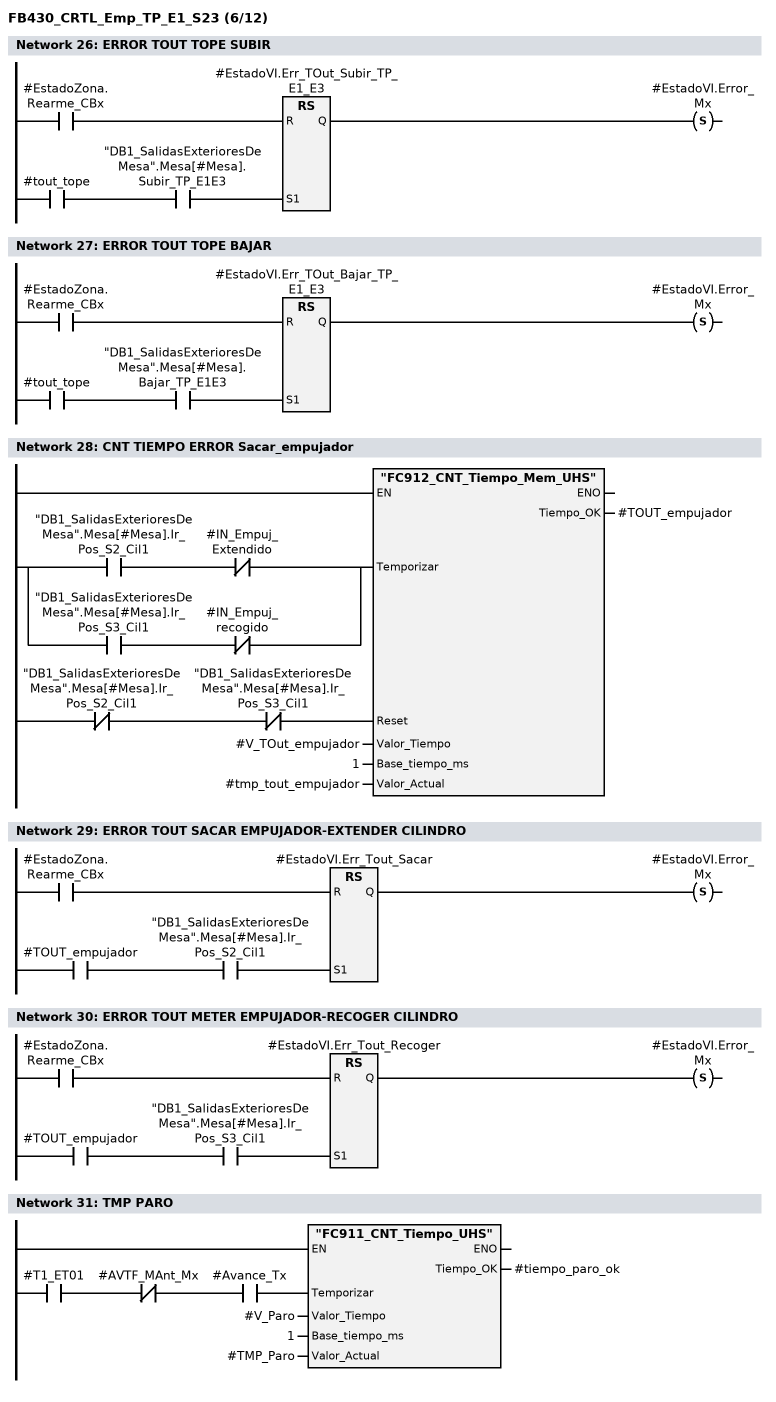
   RUNG wire#powerrail
      Contact( #EstadoZona.Rearme_CBx )
      S_RS(operand := #EstadoVI.Err_TOut_Subir_TP_E1_E3, s1 := wire#w1)
      S_Coil( #EstadoVI.Error_Mx )
   END_RUNG
   RUNG wire#powerrail
      Contact( #tout_tope )
      Contact( "DB1_SalidasExterioresDeMesa".Mesa[#Mesa].Subir_TP_E1E3 )
   END_RUNG wire#w1
   // the same network as SCL:
   IF #EstadoZona.Rearme_CBx THEN
       #EstadoVI.Err_TOut_Subir_TP_E1_E3 := FALSE;   // RS flip-flop
   END_IF;
   IF #tout_tope AND "DB1_SalidasExterioresDeMesa".Mesa[#Mesa].Subir_TP_E1E3 THEN
       #EstadoVI.Err_TOut_Subir_TP_E1_E3 := TRUE;
   END_IF;
   IF #EstadoVI.Err_TOut_Subir_TP_E1_E3 THEN #EstadoVI.Error_Mx := TRUE; END_IF;
END_REGION

REGION Network 27: ERROR TOUT TOPE BAJAR
   RUNG wire#powerrail
      Contact( #EstadoZona.Rearme_CBx )
      S_RS(operand := #EstadoVI.Err_TOut_Bajar_TP_E1_E3, s1 := wire#w1)
      S_Coil( #EstadoVI.Error_Mx )
   END_RUNG
   RUNG wire#powerrail
      Contact( #tout_tope )
      Contact( "DB1_SalidasExterioresDeMesa".Mesa[#Mesa].Bajar_TP_E1E3 )
   END_RUNG wire#w1
   // the same network as SCL:
   IF #EstadoZona.Rearme_CBx THEN
       #EstadoVI.Err_TOut_Bajar_TP_E1_E3 := FALSE;   // RS flip-flop
   END_IF;
   IF #tout_tope AND "DB1_SalidasExterioresDeMesa".Mesa[#Mesa].Bajar_TP_E1E3 THEN
       #EstadoVI.Err_TOut_Bajar_TP_E1_E3 := TRUE;
   END_IF;
   IF #EstadoVI.Err_TOut_Bajar_TP_E1_E3 THEN #EstadoVI.Error_Mx := TRUE; END_IF;
END_REGION

REGION Network 28: CNT TIEMPO ERROR Sacar_empujador
   RUNG wire#powerrail
      "FC912_CNT_Tiempo_Mem_UHS"(Temporizar := wire#w1, Reset := wire#w2, Valor_Tiempo := #V_TOut_empujador, Base_tiempo_ms := 1, Valor_Actual := #tmp_tout_empujador, Tiempo_OK => #TOUT_empujador)
   END_RUNG
   RUNG wire#powerrail
      Contact( "DB1_SalidasExterioresDeMesa".Mesa[#Mesa].Ir_Pos_S2_Cil1 )
      I_Contact( #IN_Empuj_Extendido )
   END_RUNG wire#w1
   RUNG wire#powerrail
      Contact( "DB1_SalidasExterioresDeMesa".Mesa[#Mesa].Ir_Pos_S3_Cil1 )
      I_Contact( #IN_Empuj_recogido )
   END_RUNG wire#w1
   RUNG wire#powerrail
      I_Contact( "DB1_SalidasExterioresDeMesa".Mesa[#Mesa].Ir_Pos_S2_Cil1 )
      I_Contact( "DB1_SalidasExterioresDeMesa".Mesa[#Mesa].Ir_Pos_S3_Cil1 )
   END_RUNG wire#w2
   // the same network as SCL:
   "FC912_CNT_Tiempo_Mem_UHS"(Temporizar := ("DB1_SalidasExterioresDeMesa".Mesa[#Mesa].Ir_Pos_S2_Cil1 AND NOT #IN_Empuj_Extendido) OR ("DB1_SalidasExterioresDeMesa".Mesa[#Mesa].Ir_Pos_S3_Cil1 AND NOT #IN_Empuj_recogido),
                           Reset := NOT "DB1_SalidasExterioresDeMesa".Mesa[#Mesa].Ir_Pos_S2_Cil1 AND NOT "DB1_SalidasExterioresDeMesa".Mesa[#Mesa].Ir_Pos_S3_Cil1,
                           Valor_Tiempo := #V_TOut_empujador,
                           Base_tiempo_ms := 1,
                           Valor_Actual := #tmp_tout_empujador,
                           Tiempo_OK => #TOUT_empujador);
END_REGION

REGION Network 29: ERROR TOUT SACAR EMPUJADOR-EXTENDER CILINDRO
   RUNG wire#powerrail
      Contact( #EstadoZona.Rearme_CBx )
      S_RS(operand := #EstadoVI.Err_Tout_Sacar, s1 := wire#w1)
      S_Coil( #EstadoVI.Error_Mx )
   END_RUNG
   RUNG wire#powerrail
      Contact( #TOUT_empujador )
      Contact( "DB1_SalidasExterioresDeMesa".Mesa[#Mesa].Ir_Pos_S2_Cil1 )
   END_RUNG wire#w1
   // the same network as SCL:
   IF #EstadoZona.Rearme_CBx THEN
       #EstadoVI.Err_Tout_Sacar := FALSE;   // RS flip-flop
   END_IF;
   IF #TOUT_empujador AND "DB1_SalidasExterioresDeMesa".Mesa[#Mesa].Ir_Pos_S2_Cil1 THEN
       #EstadoVI.Err_Tout_Sacar := TRUE;
   END_IF;
   IF #EstadoVI.Err_Tout_Sacar THEN #EstadoVI.Error_Mx := TRUE; END_IF;
END_REGION

REGION Network 30: ERROR TOUT METER EMPUJADOR-RECOGER CILINDRO
   RUNG wire#powerrail
      Contact( #EstadoZona.Rearme_CBx )
      S_RS(operand := #EstadoVI.Err_Tout_Recoger, s1 := wire#w1)
      S_Coil( #EstadoVI.Error_Mx )
   END_RUNG
   RUNG wire#powerrail
      Contact( #TOUT_empujador )
      Contact( "DB1_SalidasExterioresDeMesa".Mesa[#Mesa].Ir_Pos_S3_Cil1 )
   END_RUNG wire#w1
   // the same network as SCL:
   IF #EstadoZona.Rearme_CBx THEN
       #EstadoVI.Err_Tout_Recoger := FALSE;   // RS flip-flop
   END_IF;
   IF #TOUT_empujador AND "DB1_SalidasExterioresDeMesa".Mesa[#Mesa].Ir_Pos_S3_Cil1 THEN
       #EstadoVI.Err_Tout_Recoger := TRUE;
   END_IF;
   IF #EstadoVI.Err_Tout_Recoger THEN #EstadoVI.Error_Mx := TRUE; END_IF;
END_REGION

REGION Network 31: TMP PARO
   RUNG wire#powerrail
      "FC911_CNT_Tiempo_UHS"(Temporizar := wire#w1, Valor_Tiempo := #V_Paro, Base_tiempo_ms := 1, Valor_Actual := #TMP_Paro, Tiempo_OK => #tiempo_paro_ok)
   END_RUNG
   RUNG wire#powerrail
      Contact( #T1_ET01 )
      I_Contact( #AVTF_MAnt_Mx )
      Contact( #Avance_Tx )
   END_RUNG wire#w1
   // the same network as SCL:
   "FC911_CNT_Tiempo_UHS"(Temporizar := #T1_ET01 AND NOT #AVTF_MAnt_Mx AND #Avance_Tx,
                          Valor_Tiempo := #V_Paro,
                          Base_tiempo_ms := 1,
                          Valor_Actual := #TMP_Paro,
                          Tiempo_OK => #tiempo_paro_ok);
END_REGION

REGION Network 32: Vaciado y tiempo Maximo espera orden Scanner
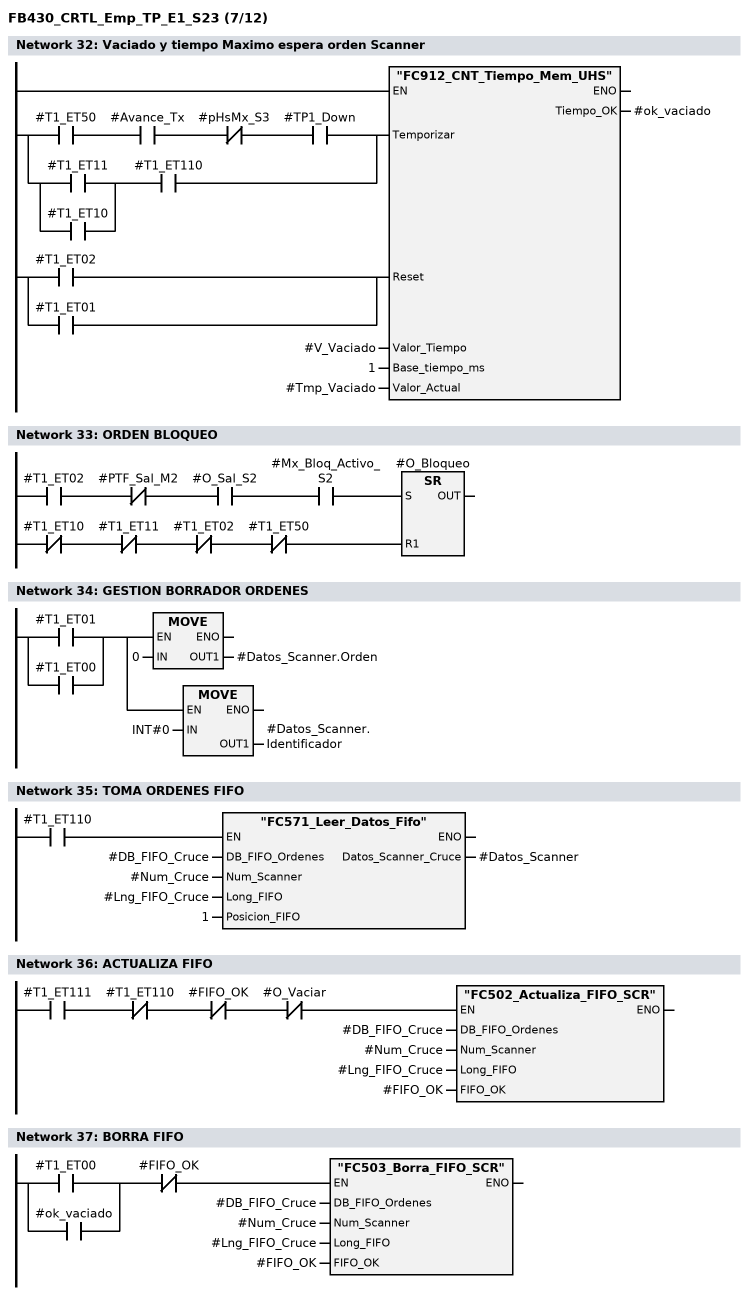
   RUNG wire#powerrail
      "FC912_CNT_Tiempo_Mem_UHS"(Temporizar := wire#w2, Reset := wire#w3, Valor_Tiempo := #V_Vaciado, Base_tiempo_ms := 1, Valor_Actual := #Tmp_Vaciado, Tiempo_OK => #ok_vaciado)
   END_RUNG
   RUNG wire#powerrail
      Contact( #T1_ET50 )
      Contact( #Avance_Tx )
      I_Contact( #pHsMx_S3 )
      Contact( #TP1_Down )
   END_RUNG wire#w2
   RUNG wire#powerrail
      Contact( #T1_ET11 )
      wire#w1
      Contact( #T1_ET110 )
   END_RUNG wire#w2
   RUNG wire#powerrail
      Contact( #T1_ET10 )
   END_RUNG wire#w1
   RUNG wire#powerrail
      Contact( #T1_ET02 )
   END_RUNG wire#w3
   RUNG wire#powerrail
      Contact( #T1_ET01 )
   END_RUNG wire#w3
   // the same network as SCL:
   "FC912_CNT_Tiempo_Mem_UHS"(Temporizar := (#T1_ET50 AND #Avance_Tx AND NOT #pHsMx_S3 AND #TP1_Down) OR ((#T1_ET11 OR #T1_ET10) AND #T1_ET110),
                           Reset := #T1_ET02 OR #T1_ET01,
                           Valor_Tiempo := #V_Vaciado,
                           Base_tiempo_ms := 1,
                           Valor_Actual := #Tmp_Vaciado,
                           Tiempo_OK => #ok_vaciado);
END_REGION

REGION Network 33: ORDEN BLOQUEO
   RUNG wire#powerrail
      Contact( #T1_ET02 )
      I_Contact( #PTF_Sal_M2 )
      Contact( #O_Sal_S2 )
      Contact( #Mx_Bloq_Activo_S2 )
      S_SR(operand := #O_Bloqueo, r1 := wire#w1)
   END_RUNG
   RUNG wire#powerrail
      I_Contact( #T1_ET10 )
      I_Contact( #T1_ET11 )
      I_Contact( #T1_ET02 )
      I_Contact( #T1_ET50 )
   END_RUNG wire#w1
   // the same network as SCL:
   IF #T1_ET02 AND NOT #PTF_Sal_M2 AND #O_Sal_S2 AND #Mx_Bloq_Activo_S2 THEN
       #O_Bloqueo := TRUE;   // SR flip-flop
   END_IF;
   IF NOT #T1_ET10 AND NOT #T1_ET11 AND NOT #T1_ET02 AND NOT #T1_ET50 THEN #O_Bloqueo := FALSE; END_IF;
END_REGION

REGION Network 34: GESTION BORRADOR ORDENES
   RUNG wire#powerrail
      Contact( #T1_ET01 )
      wire#w1
      { S7_GenerateENO := "TRUE" } Move(in := 0, out1 => #Datos_Scanner.Orden)
   END_RUNG
   RUNG wire#powerrail
      Contact( #T1_ET00 )
   END_RUNG wire#w1
   RUNG wire#w1
      { S7_GenerateENO := "TRUE" } Move(in := INT#0, out1 => #Datos_Scanner.Identificador)
   END_RUNG
   // the same network as SCL:
   IF #T1_ET01 OR #T1_ET00 THEN
       #Datos_Scanner.Orden := 0;
       #Datos_Scanner.Identificador := INT#0;
   END_IF;
END_REGION

REGION Network 35: TOMA ORDENES FIFO
   RUNG wire#powerrail
      Contact( #T1_ET110 )
      "FC571_Leer_Datos_Fifo"(DB_FIFO_Ordenes := #DB_FIFO_Cruce, Num_Scanner := #Num_Cruce, Long_FIFO := #Lng_FIFO_Cruce, Posicion_FIFO := 1, Datos_Scanner_Cruce => #Datos_Scanner)
   END_RUNG
   // the same network as SCL:
   IF #T1_ET110 THEN
       "FC571_Leer_Datos_Fifo"(DB_FIFO_Ordenes := #DB_FIFO_Cruce,
                               Num_Scanner := #Num_Cruce,
                               Long_FIFO := #Lng_FIFO_Cruce,
                               Posicion_FIFO := 1,
                               Datos_Scanner_Cruce => #Datos_Scanner);
   END_IF;
END_REGION

REGION Network 36: ACTUALIZA FIFO
   RUNG wire#powerrail
      Contact( #T1_ET111 )
      I_Contact( #T1_ET110 )
      I_Contact( #FIFO_OK )
      I_Contact( #O_Vaciar )
      "FC502_Actualiza_FIFO_SCR"(DB_FIFO_Ordenes := #DB_FIFO_Cruce, Num_Scanner := #Num_Cruce, Long_FIFO := #Lng_FIFO_Cruce, FIFO_OK := #FIFO_OK)
   END_RUNG
   // the same network as SCL:
   IF #T1_ET111 AND NOT #T1_ET110 AND NOT #FIFO_OK AND NOT #O_Vaciar THEN
       "FC502_Actualiza_FIFO_SCR"(DB_FIFO_Ordenes := #DB_FIFO_Cruce,
                               Num_Scanner := #Num_Cruce,
                               Long_FIFO := #Lng_FIFO_Cruce,
                               FIFO_OK := #FIFO_OK);
   END_IF;
END_REGION

REGION Network 37: BORRA FIFO
   RUNG wire#powerrail
      Contact( #T1_ET00 )
      wire#w1
      I_Contact( #FIFO_OK )
      "FC503_Borra_FIFO_SCR"(DB_FIFO_Ordenes := #DB_FIFO_Cruce, Num_Scanner := #Num_Cruce, Long_FIFO := #Lng_FIFO_Cruce, FIFO_OK := #FIFO_OK)
   END_RUNG
   RUNG wire#powerrail
      Contact( #ok_vaciado )
   END_RUNG wire#w1
   // the same network as SCL:
   IF (#T1_ET00 OR #ok_vaciado) AND NOT #FIFO_OK THEN
       "FC503_Borra_FIFO_SCR"(DB_FIFO_Ordenes := #DB_FIFO_Cruce,
                              Num_Scanner := #Num_Cruce,
                              Long_FIFO := #Lng_FIFO_Cruce,
                              FIFO_OK := #FIFO_OK);
   END_IF;
END_REGION

REGION Network 38: PASAR ORDEN S3
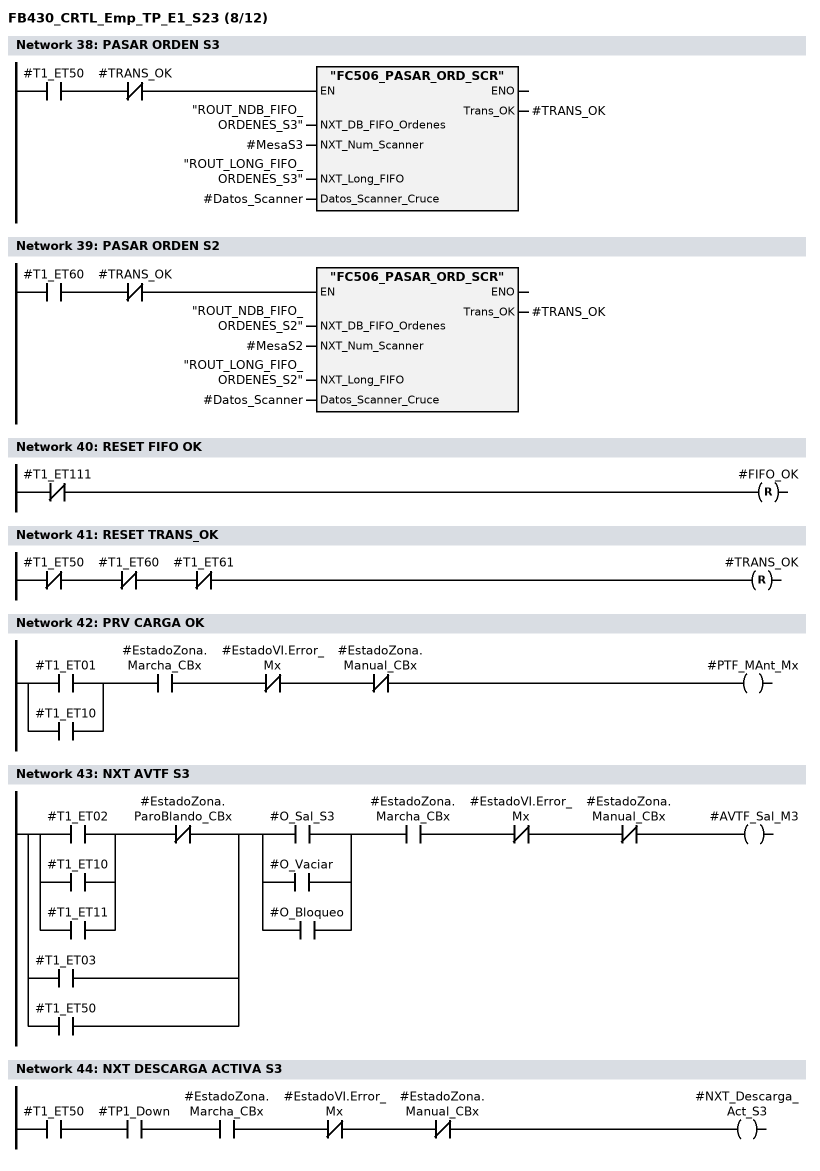
   RUNG wire#powerrail
      Contact( #T1_ET50 )
      I_Contact( #TRANS_OK )
      "FC506_PASAR_ORD_SCR"(NXT_DB_FIFO_Ordenes := "ROUT_NDB_FIFO_ORDENES_S3", NXT_Num_Scanner := #MesaS3, NXT_Long_FIFO := "ROUT_LONG_FIFO_ORDENES_S3", Datos_Scanner_Cruce := #Datos_Scanner, Trans_OK => #TRANS_OK)
   END_RUNG
   // the same network as SCL:
   IF #T1_ET50 AND NOT #TRANS_OK THEN
       "FC506_PASAR_ORD_SCR"(NXT_DB_FIFO_Ordenes := "ROUT_NDB_FIFO_ORDENES_S3",
                             NXT_Num_Scanner := #MesaS3,
                             NXT_Long_FIFO := "ROUT_LONG_FIFO_ORDENES_S3",
                             Datos_Scanner_Cruce := #Datos_Scanner,
                             Trans_OK => #TRANS_OK);
   END_IF;
END_REGION

REGION Network 39: PASAR ORDEN S2
   RUNG wire#powerrail
      Contact( #T1_ET60 )
      I_Contact( #TRANS_OK )
      "FC506_PASAR_ORD_SCR"(NXT_DB_FIFO_Ordenes := "ROUT_NDB_FIFO_ORDENES_S2", NXT_Num_Scanner := #MesaS2, NXT_Long_FIFO := "ROUT_LONG_FIFO_ORDENES_S2", Datos_Scanner_Cruce := #Datos_Scanner, Trans_OK => #TRANS_OK)
   END_RUNG
   // the same network as SCL:
   IF #T1_ET60 AND NOT #TRANS_OK THEN
       "FC506_PASAR_ORD_SCR"(NXT_DB_FIFO_Ordenes := "ROUT_NDB_FIFO_ORDENES_S2",
                             NXT_Num_Scanner := #MesaS2,
                             NXT_Long_FIFO := "ROUT_LONG_FIFO_ORDENES_S2",
                             Datos_Scanner_Cruce := #Datos_Scanner,
                             Trans_OK => #TRANS_OK);
   END_IF;
END_REGION

REGION Network 40: RESET FIFO OK
   RUNG wire#powerrail
      I_Contact( #T1_ET111 )
      R_Coil( #FIFO_OK )
   END_RUNG
   // the same network as SCL:
   IF NOT #T1_ET111 THEN #FIFO_OK := FALSE; END_IF;
END_REGION

REGION Network 41: RESET TRANS_OK
   RUNG wire#powerrail
      I_Contact( #T1_ET50 )
      I_Contact( #T1_ET60 )
      I_Contact( #T1_ET61 )
      R_Coil( #TRANS_OK )
   END_RUNG
   // the same network as SCL:
   IF NOT #T1_ET50 AND NOT #T1_ET60 AND NOT #T1_ET61 THEN #TRANS_OK := FALSE; END_IF;
END_REGION

REGION Network 42: PRV CARGA OK
   RUNG wire#powerrail
      Contact( #T1_ET01 )
      wire#w1
      Contact( #EstadoZona.Marcha_CBx )
      I_Contact( #EstadoVI.Error_Mx )
      I_Contact( #EstadoZona.Manual_CBx )
      Coil( #PTF_MAnt_Mx )
   END_RUNG
   RUNG wire#powerrail
      Contact( #T1_ET10 )
   END_RUNG wire#w1
   // the same network as SCL:
   #PTF_MAnt_Mx := (#T1_ET01 OR #T1_ET10) AND #EstadoZona.Marcha_CBx AND NOT #EstadoVI.Error_Mx AND NOT #EstadoZona.Manual_CBx;
END_REGION

REGION Network 43: NXT AVTF S3
   RUNG wire#powerrail
      Contact( #T1_ET02 )
      wire#w1
      I_Contact( #EstadoZona.ParoBlando_CBx )
      wire#w2
      Contact( #O_Sal_S3 )
      wire#w3
      Contact( #EstadoZona.Marcha_CBx )
      I_Contact( #EstadoVI.Error_Mx )
      I_Contact( #EstadoZona.Manual_CBx )
      Coil( #AVTF_Sal_M3 )
   END_RUNG
   RUNG wire#powerrail
      Contact( #T1_ET10 )
   END_RUNG wire#w1
   RUNG wire#powerrail
      Contact( #T1_ET11 )
   END_RUNG wire#w1
   RUNG wire#powerrail
      Contact( #T1_ET03 )
   END_RUNG wire#w2
   RUNG wire#powerrail
      Contact( #T1_ET50 )
   END_RUNG wire#w2
   RUNG wire#w2
      Contact( #O_Vaciar )
   END_RUNG wire#w3
   RUNG wire#w2
      Contact( #O_Bloqueo )
   END_RUNG wire#w3
   // the same network as SCL:
   #AVTF_Sal_M3 := (((#T1_ET02 OR #T1_ET10 OR #T1_ET11) AND NOT #EstadoZona.ParoBlando_CBx) OR #T1_ET03 OR #T1_ET50) AND (#O_Sal_S3 OR #O_Vaciar OR #O_Bloqueo) AND #EstadoZona.Marcha_CBx AND NOT #EstadoVI.Error_Mx AND NOT #EstadoZona.Manual_CBx;
END_REGION

REGION Network 44: NXT DESCARGA ACTIVA S3
   RUNG wire#powerrail
      Contact( #T1_ET50 )
      Contact( #TP1_Down )
      Contact( #EstadoZona.Marcha_CBx )
      I_Contact( #EstadoVI.Error_Mx )
      I_Contact( #EstadoZona.Manual_CBx )
      Coil( #NXT_Descarga_Act_S3 )
   END_RUNG
   // the same network as SCL:
   #NXT_Descarga_Act_S3 := #T1_ET50 AND #TP1_Down AND #EstadoZona.Marcha_CBx AND NOT #EstadoVI.Error_Mx AND NOT #EstadoZona.Manual_CBx;
END_REGION

REGION Network 45: NXT AVTF S2
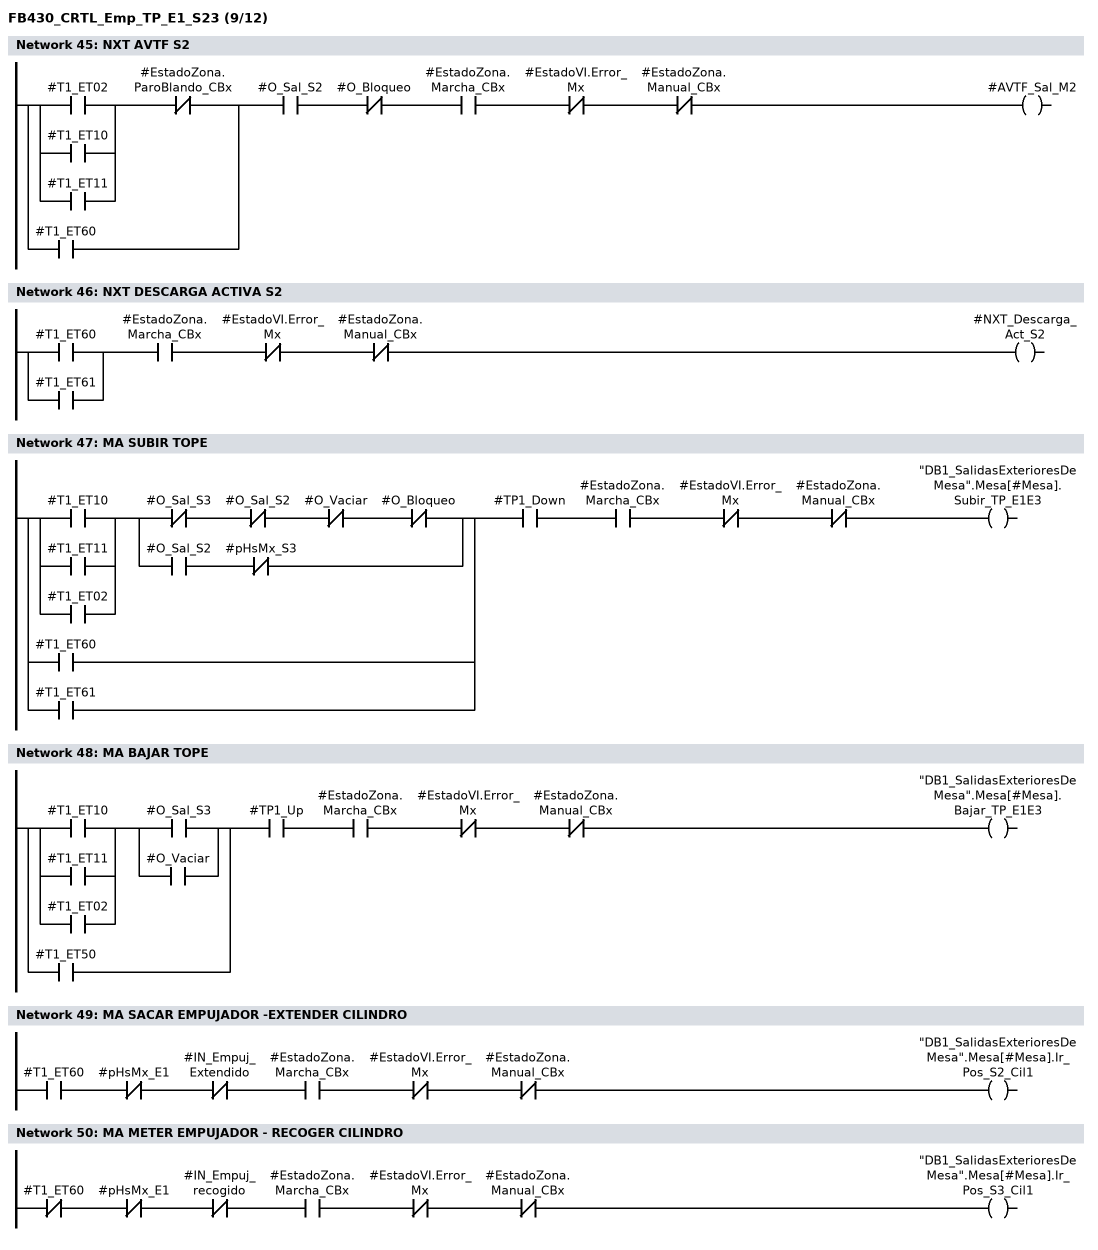
   RUNG wire#powerrail
      Contact( #T1_ET02 )
      wire#w1
      I_Contact( #EstadoZona.ParoBlando_CBx )
      wire#w2
      Contact( #O_Sal_S2 )
      I_Contact( #O_Bloqueo )
      Contact( #EstadoZona.Marcha_CBx )
      I_Contact( #EstadoVI.Error_Mx )
      I_Contact( #EstadoZona.Manual_CBx )
      Coil( #AVTF_Sal_M2 )
   END_RUNG
   RUNG wire#powerrail
      Contact( #T1_ET10 )
   END_RUNG wire#w1
   RUNG wire#powerrail
      Contact( #T1_ET11 )
   END_RUNG wire#w1
   RUNG wire#powerrail
      Contact( #T1_ET60 )
   END_RUNG wire#w2
   // the same network as SCL:
   #AVTF_Sal_M2 := (((#T1_ET02 OR #T1_ET10 OR #T1_ET11) AND NOT #EstadoZona.ParoBlando_CBx) OR #T1_ET60) AND #O_Sal_S2 AND NOT #O_Bloqueo AND #EstadoZona.Marcha_CBx AND NOT #EstadoVI.Error_Mx AND NOT #EstadoZona.Manual_CBx;
END_REGION

REGION Network 46: NXT DESCARGA ACTIVA S2
   RUNG wire#powerrail
      Contact( #T1_ET60 )
      wire#w1
      Contact( #EstadoZona.Marcha_CBx )
      I_Contact( #EstadoVI.Error_Mx )
      I_Contact( #EstadoZona.Manual_CBx )
      Coil( #NXT_Descarga_Act_S2 )
   END_RUNG
   RUNG wire#powerrail
      Contact( #T1_ET61 )
   END_RUNG wire#w1
   // the same network as SCL:
   #NXT_Descarga_Act_S2 := (#T1_ET60 OR #T1_ET61) AND #EstadoZona.Marcha_CBx AND NOT #EstadoVI.Error_Mx AND NOT #EstadoZona.Manual_CBx;
END_REGION

REGION Network 47: MA SUBIR TOPE
   RUNG wire#powerrail
      Contact( #T1_ET10 )
      wire#w1
      I_Contact( #O_Sal_S3 )
      I_Contact( #O_Sal_S2 )
      I_Contact( #O_Vaciar )
      I_Contact( #O_Bloqueo )
      wire#w2
      Contact( #TP1_Down )
      Contact( #EstadoZona.Marcha_CBx )
      I_Contact( #EstadoVI.Error_Mx )
      I_Contact( #EstadoZona.Manual_CBx )
      Coil( "DB1_SalidasExterioresDeMesa".Mesa[#Mesa].Subir_TP_E1E3 )
   END_RUNG
   RUNG wire#powerrail
      Contact( #T1_ET11 )
   END_RUNG wire#w1
   RUNG wire#powerrail
      Contact( #T1_ET02 )
   END_RUNG wire#w1
   RUNG wire#w1
      Contact( #O_Sal_S2 )
      I_Contact( #pHsMx_S3 )
   END_RUNG wire#w2
   RUNG wire#powerrail
      Contact( #T1_ET60 )
   END_RUNG wire#w2
   RUNG wire#powerrail
      Contact( #T1_ET61 )
   END_RUNG wire#w2
   // the same network as SCL:
   "DB1_SalidasExterioresDeMesa".Mesa[#Mesa].Subir_TP_E1E3 := (((#T1_ET10 OR #T1_ET11 OR #T1_ET02) AND ((NOT #O_Sal_S3 AND NOT #O_Sal_S2 AND NOT #O_Vaciar AND NOT #O_Bloqueo) OR (#O_Sal_S2 AND NOT #pHsMx_S3))) OR #T1_ET60 OR #T1_ET61) AND #TP1_Down AND #EstadoZona.Marcha_CBx AND NOT #EstadoVI.Error_Mx AND NOT #EstadoZona.Manual_CBx;
END_REGION

REGION Network 48: MA BAJAR TOPE
   RUNG wire#powerrail
      Contact( #T1_ET10 )
      wire#w1
      Contact( #O_Sal_S3 )
      wire#w2
      Contact( #TP1_Up )
      Contact( #EstadoZona.Marcha_CBx )
      I_Contact( #EstadoVI.Error_Mx )
      I_Contact( #EstadoZona.Manual_CBx )
      Coil( "DB1_SalidasExterioresDeMesa".Mesa[#Mesa].Bajar_TP_E1E3 )
   END_RUNG
   RUNG wire#powerrail
      Contact( #T1_ET11 )
   END_RUNG wire#w1
   RUNG wire#powerrail
      Contact( #T1_ET02 )
   END_RUNG wire#w1
   RUNG wire#w1
      Contact( #O_Vaciar )
   END_RUNG wire#w2
   RUNG wire#powerrail
      Contact( #T1_ET50 )
   END_RUNG wire#w2
   // the same network as SCL:
   "DB1_SalidasExterioresDeMesa".Mesa[#Mesa].Bajar_TP_E1E3 := (((#T1_ET10 OR #T1_ET11 OR #T1_ET02) AND (#O_Sal_S3 OR #O_Vaciar)) OR #T1_ET50) AND #TP1_Up AND #EstadoZona.Marcha_CBx AND NOT #EstadoVI.Error_Mx AND NOT #EstadoZona.Manual_CBx;
END_REGION

REGION Network 49: MA SACAR EMPUJADOR -EXTENDER CILINDRO
   RUNG wire#powerrail
      Contact( #T1_ET60 )
      I_Contact( #pHsMx_E1 )
      I_Contact( #IN_Empuj_Extendido )
      Contact( #EstadoZona.Marcha_CBx )
      I_Contact( #EstadoVI.Error_Mx )
      I_Contact( #EstadoZona.Manual_CBx )
      Coil( "DB1_SalidasExterioresDeMesa".Mesa[#Mesa].Ir_Pos_S2_Cil1 )
   END_RUNG
   // the same network as SCL:
   "DB1_SalidasExterioresDeMesa".Mesa[#Mesa].Ir_Pos_S2_Cil1 := #T1_ET60 AND NOT #pHsMx_E1 AND NOT #IN_Empuj_Extendido AND #EstadoZona.Marcha_CBx AND NOT #EstadoVI.Error_Mx AND NOT #EstadoZona.Manual_CBx;
END_REGION

REGION Network 50: MA METER EMPUJADOR - RECOGER CILINDRO
   RUNG wire#powerrail
      I_Contact( #T1_ET60 )
      I_Contact( #pHsMx_E1 )
      I_Contact( #IN_Empuj_recogido )
      Contact( #EstadoZona.Marcha_CBx )
      I_Contact( #EstadoVI.Error_Mx )
      I_Contact( #EstadoZona.Manual_CBx )
      Coil( "DB1_SalidasExterioresDeMesa".Mesa[#Mesa].Ir_Pos_S3_Cil1 )
   END_RUNG
   // the same network as SCL:
   "DB1_SalidasExterioresDeMesa".Mesa[#Mesa].Ir_Pos_S3_Cil1 := NOT #T1_ET60 AND NOT #pHsMx_E1 AND NOT #IN_Empuj_recogido AND #EstadoZona.Marcha_CBx AND NOT #EstadoVI.Error_Mx AND NOT #EstadoZona.Manual_CBx;
END_REGION

REGION Network 51: MA AVANCE 13
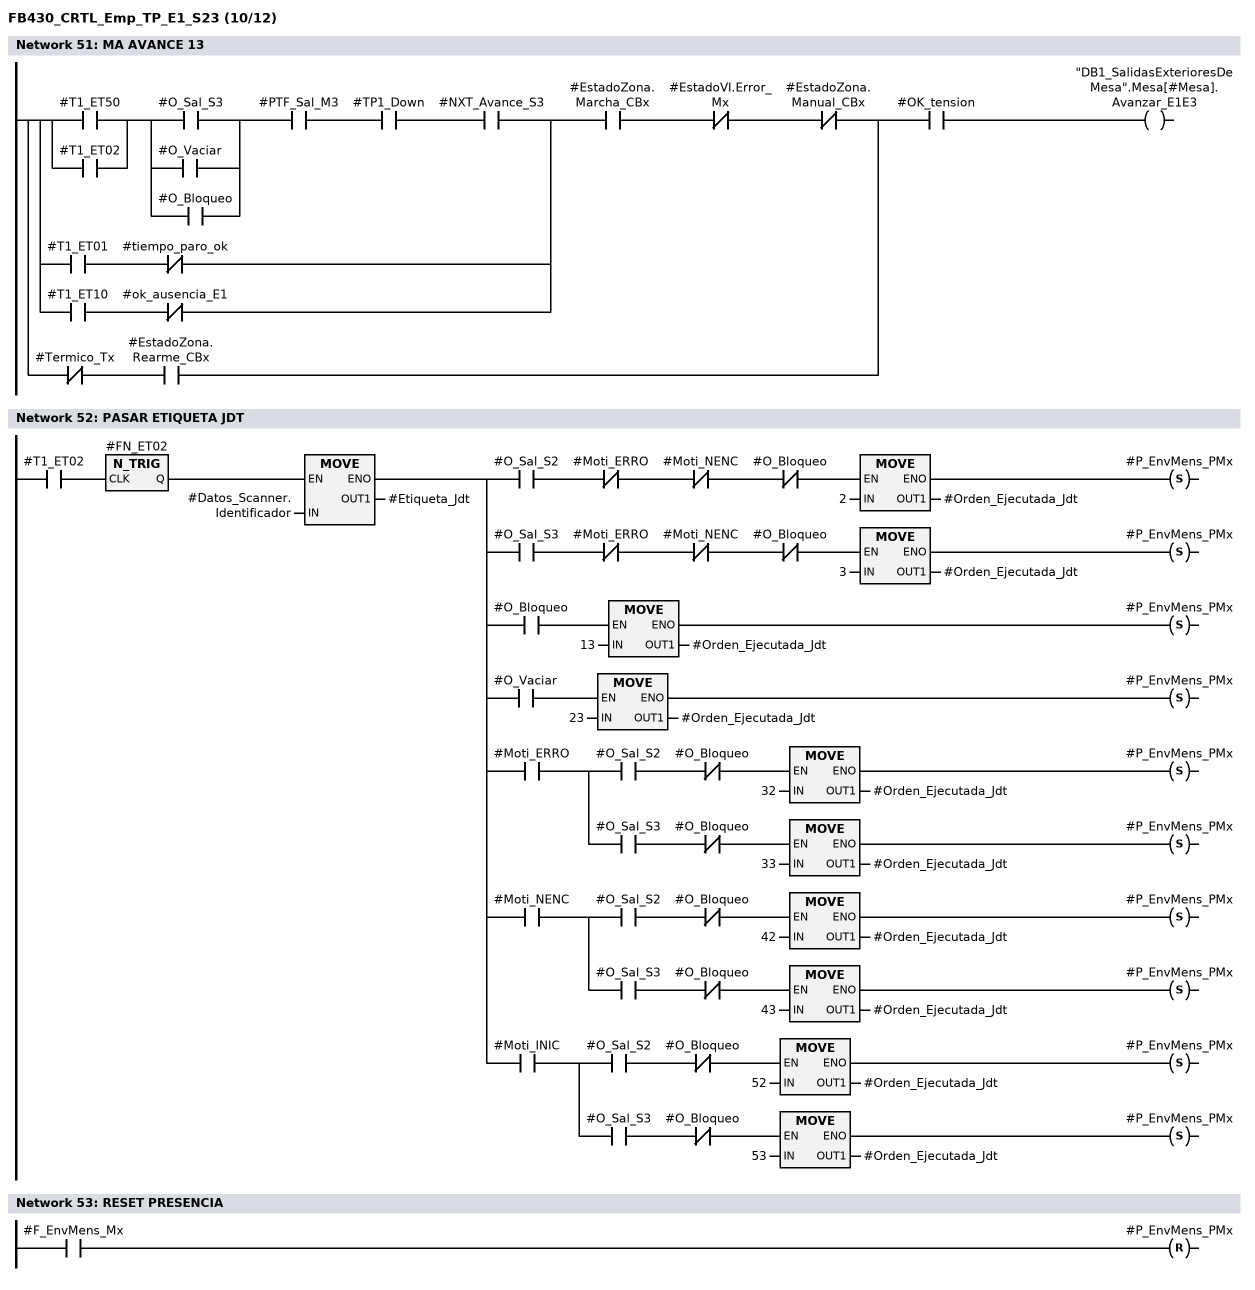
   RUNG wire#powerrail
      Contact( #T1_ET50 )
      wire#w1
      Contact( #O_Sal_S3 )
      wire#w2
      Contact( #PTF_Sal_M3 )
      Contact( #TP1_Down )
      Contact( #NXT_Avance_S3 )
      wire#w3
      Contact( #EstadoZona.Marcha_CBx )
      I_Contact( #EstadoVI.Error_Mx )
      I_Contact( #EstadoZona.Manual_CBx )
      wire#w4
      Contact( #OK_tension )
      Coil( "DB1_SalidasExterioresDeMesa".Mesa[#Mesa].Avanzar_E1E3 )
   END_RUNG
   RUNG wire#powerrail
      Contact( #T1_ET02 )
   END_RUNG wire#w1
   RUNG wire#w1
      Contact( #O_Vaciar )
   END_RUNG wire#w2
   RUNG wire#w1
      Contact( #O_Bloqueo )
   END_RUNG wire#w2
   RUNG wire#powerrail
      Contact( #T1_ET01 )
      I_Contact( #tiempo_paro_ok )
   END_RUNG wire#w3
   RUNG wire#powerrail
      Contact( #T1_ET10 )
      I_Contact( #ok_ausencia_E1 )
   END_RUNG wire#w3
   RUNG wire#powerrail
      I_Contact( #Termico_Tx )
      Contact( #EstadoZona.Rearme_CBx )
   END_RUNG wire#w4
   // the same network as SCL:
   "DB1_SalidasExterioresDeMesa".Mesa[#Mesa].Avanzar_E1E3 := (((((#T1_ET50 OR #T1_ET02) AND (#O_Sal_S3 OR #O_Vaciar OR #O_Bloqueo) AND #PTF_Sal_M3 AND #TP1_Down AND #NXT_Avance_S3) OR (#T1_ET01 AND NOT #tiempo_paro_ok) OR (#T1_ET10 AND NOT #ok_ausencia_E1)) AND #EstadoZona.Marcha_CBx AND NOT #EstadoVI.Error_Mx AND NOT #EstadoZona.Manual_CBx) OR (NOT #Termico_Tx AND #EstadoZona.Rearme_CBx)) AND #OK_tension;
END_REGION

REGION Network 52: PASAR ETIQUETA JDT
   RUNG wire#powerrail
      Contact( #T1_ET02 )
      N_Trig( #FN_ET02 )
      { S7_GenerateENO := "TRUE" } Move(in := #Datos_Scanner.Identificador, out1 => #Etiqueta_Jdt)
      wire#w1
      Contact( #O_Sal_S2 )
      I_Contact( #Moti_ERRO )
      I_Contact( #Moti_NENC )
      I_Contact( #O_Bloqueo )
      { S7_GenerateENO := "TRUE" } Move(in := 2, out1 => #Orden_Ejecutada_Jdt)
      S_Coil( #P_EnvMens_PMx )
   END_RUNG
   RUNG wire#w1
      Contact( #O_Sal_S3 )
      I_Contact( #Moti_ERRO )
      I_Contact( #Moti_NENC )
      I_Contact( #O_Bloqueo )
      { S7_GenerateENO := "TRUE" } Move(in := 3, out1 => #Orden_Ejecutada_Jdt)
      S_Coil( #P_EnvMens_PMx )
   END_RUNG
   RUNG wire#w1
      Contact( #O_Bloqueo )
      { S7_GenerateENO := "TRUE" } Move(in := 13, out1 => #Orden_Ejecutada_Jdt)
      S_Coil( #P_EnvMens_PMx )
   END_RUNG
   RUNG wire#w1
      Contact( #O_Vaciar )
      { S7_GenerateENO := "TRUE" } Move(in := 23, out1 => #Orden_Ejecutada_Jdt)
      S_Coil( #P_EnvMens_PMx )
   END_RUNG
   RUNG wire#w1
      Contact( #Moti_ERRO )
      wire#w2
      Contact( #O_Sal_S2 )
      I_Contact( #O_Bloqueo )
      { S7_GenerateENO := "TRUE" } Move(in := 32, out1 => #Orden_Ejecutada_Jdt)
      S_Coil( #P_EnvMens_PMx )
   END_RUNG
   RUNG wire#w2
      Contact( #O_Sal_S3 )
      I_Contact( #O_Bloqueo )
      { S7_GenerateENO := "TRUE" } Move(in := 33, out1 => #Orden_Ejecutada_Jdt)
      S_Coil( #P_EnvMens_PMx )
   END_RUNG
   RUNG wire#w1
      Contact( #Moti_NENC )
      wire#w3
      Contact( #O_Sal_S2 )
      I_Contact( #O_Bloqueo )
      { S7_GenerateENO := "TRUE" } Move(in := 42, out1 => #Orden_Ejecutada_Jdt)
      S_Coil( #P_EnvMens_PMx )
   END_RUNG
   RUNG wire#w3
      Contact( #O_Sal_S3 )
      I_Contact( #O_Bloqueo )
      { S7_GenerateENO := "TRUE" } Move(in := 43, out1 => #Orden_Ejecutada_Jdt)
      S_Coil( #P_EnvMens_PMx )
   END_RUNG
   RUNG wire#w1
      Contact( #Moti_INIC )
      wire#w4
      Contact( #O_Sal_S2 )
      I_Contact( #O_Bloqueo )
      { S7_GenerateENO := "TRUE" } Move(in := 52, out1 => #Orden_Ejecutada_Jdt)
      S_Coil( #P_EnvMens_PMx )
   END_RUNG
   RUNG wire#w4
      Contact( #O_Sal_S3 )
      I_Contact( #O_Bloqueo )
      { S7_GenerateENO := "TRUE" } Move(in := 53, out1 => #Orden_Ejecutada_Jdt)
      S_Coil( #P_EnvMens_PMx )
   END_RUNG
   // the same network as SCL:
   // ENO of a box is taken as its EN; it also drops when the box reports an error
   #_w1 := NOT #T1_ET02 AND #FN_ET02;   // falling edge
   #FN_ET02 := #T1_ET02;
   IF #_w1 THEN #Etiqueta_Jdt := #Datos_Scanner.Identificador; END_IF;
   IF #_w1 AND #O_Sal_S2 AND NOT #Moti_ERRO AND NOT #Moti_NENC AND NOT #O_Bloqueo THEN
       #Orden_Ejecutada_Jdt := 2;
       #P_EnvMens_PMx := TRUE;
   END_IF;
   IF #_w1 AND #O_Sal_S3 AND NOT #Moti_ERRO AND NOT #Moti_NENC AND NOT #O_Bloqueo THEN
       #Orden_Ejecutada_Jdt := 3;
       #P_EnvMens_PMx := TRUE;
   END_IF;
   IF #_w1 AND #O_Bloqueo THEN
       #Orden_Ejecutada_Jdt := 13;
       #P_EnvMens_PMx := TRUE;
   END_IF;
   IF #_w1 AND #O_Vaciar THEN
       #Orden_Ejecutada_Jdt := 23;
       #P_EnvMens_PMx := TRUE;
   END_IF;
   #_w2 := #_w1 AND #Moti_ERRO;
   IF #_w2 AND #O_Sal_S2 AND NOT #O_Bloqueo THEN
       #Orden_Ejecutada_Jdt := 32;
       #P_EnvMens_PMx := TRUE;
   END_IF;
   IF #_w2 AND #O_Sal_S3 AND NOT #O_Bloqueo THEN
       #Orden_Ejecutada_Jdt := 33;
       #P_EnvMens_PMx := TRUE;
   END_IF;
   #_w3 := #_w1 AND #Moti_NENC;
   IF #_w3 AND #O_Sal_S2 AND NOT #O_Bloqueo THEN
       #Orden_Ejecutada_Jdt := 42;
       #P_EnvMens_PMx := TRUE;
   END_IF;
   IF #_w3 AND #O_Sal_S3 AND NOT #O_Bloqueo THEN
       #Orden_Ejecutada_Jdt := 43;
       #P_EnvMens_PMx := TRUE;
   END_IF;
   #_w4 := #_w1 AND #Moti_INIC;
   IF #_w4 AND #O_Sal_S2 AND NOT #O_Bloqueo THEN
       #Orden_Ejecutada_Jdt := 52;
       #P_EnvMens_PMx := TRUE;
   END_IF;
   IF #_w4 AND #O_Sal_S3 AND NOT #O_Bloqueo THEN
       #Orden_Ejecutada_Jdt := 53;
       #P_EnvMens_PMx := TRUE;
   END_IF;
END_REGION

REGION Network 53: RESET PRESENCIA
   RUNG wire#powerrail
      Contact( #F_EnvMens_Mx )
      R_Coil( #P_EnvMens_PMx )
   END_RUNG
   // the same network as SCL:
   IF #F_EnvMens_Mx THEN #P_EnvMens_PMx := FALSE; END_IF;
END_REGION

REGION Network 54: ESTADOS MESA 1
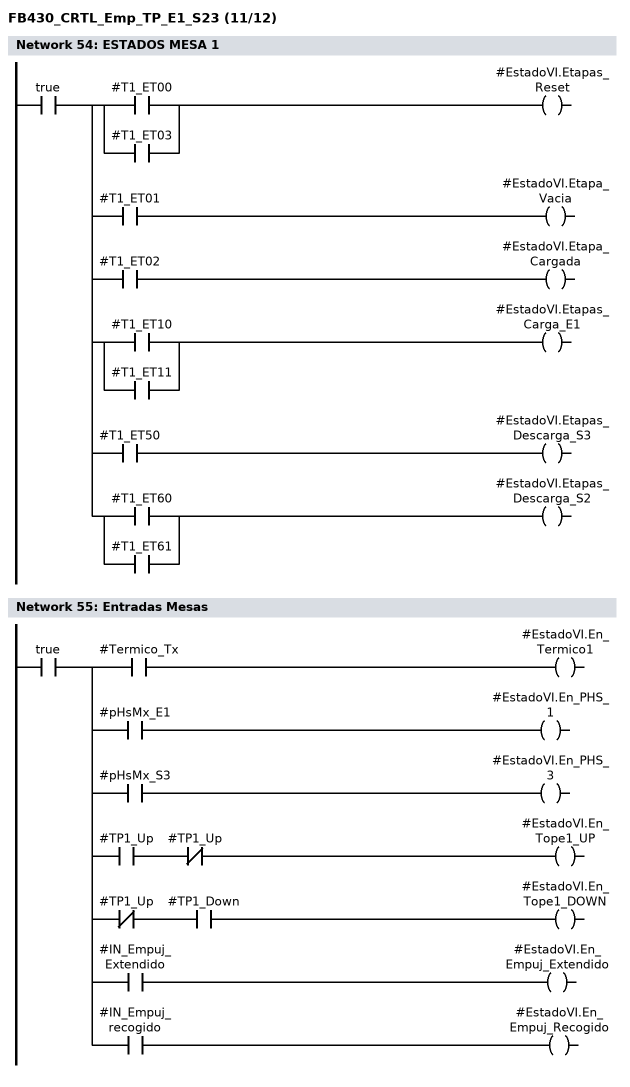
   RUNG wire#powerrail
      Contact( true )
      wire#w1
      Contact( #T1_ET00 )
      wire#w2
      Coil( #EstadoVI.Etapas_Reset )
   END_RUNG
   RUNG wire#w1
      Contact( #T1_ET03 )
   END_RUNG wire#w2
   RUNG wire#w1
      Contact( #T1_ET01 )
      Coil( #EstadoVI.Etapa_Vacia )
   END_RUNG
   RUNG wire#w1
      Contact( #T1_ET02 )
      Coil( #EstadoVI.Etapa_Cargada )
   END_RUNG
   RUNG wire#w1
      Contact( #T1_ET10 )
      wire#w3
      Coil( #EstadoVI.Etapas_Carga_E1 )
   END_RUNG
   RUNG wire#w1
      Contact( #T1_ET11 )
   END_RUNG wire#w3
   RUNG wire#w1
      Contact( #T1_ET50 )
      Coil( #EstadoVI.Etapas_Descarga_S3 )
   END_RUNG
   RUNG wire#w1
      Contact( #T1_ET60 )
      wire#w4
      Coil( #EstadoVI.Etapas_Descarga_S2 )
   END_RUNG
   RUNG wire#w1
      Contact( #T1_ET61 )
   END_RUNG wire#w4
   // the same network as SCL:
   #EstadoVI.Etapas_Reset := true AND (#T1_ET00 OR #T1_ET03);
   #EstadoVI.Etapa_Vacia := true AND #T1_ET01;
   #EstadoVI.Etapa_Cargada := true AND #T1_ET02;
   #EstadoVI.Etapas_Carga_E1 := true AND (#T1_ET10 OR #T1_ET11);
   #EstadoVI.Etapas_Descarga_S3 := true AND #T1_ET50;
   #EstadoVI.Etapas_Descarga_S2 := true AND (#T1_ET60 OR #T1_ET61);
END_REGION

REGION Network 55: Entradas Mesas
   RUNG wire#powerrail
      Contact( true )
      wire#w1
      Contact( #Termico_Tx )
      Coil( #EstadoVI.En_Termico1 )
   END_RUNG
   RUNG wire#w1
      Contact( #pHsMx_E1 )
      Coil( #EstadoVI.En_PHS_1 )
   END_RUNG
   RUNG wire#w1
      Contact( #pHsMx_S3 )
      Coil( #EstadoVI.En_PHS_3 )
   END_RUNG
   RUNG wire#w1
      Contact( #TP1_Up )
      I_Contact( #TP1_Up )
      Coil( #EstadoVI.En_Tope1_UP )
   END_RUNG
   RUNG wire#w1
      I_Contact( #TP1_Up )
      Contact( #TP1_Down )
      Coil( #EstadoVI.En_Tope1_DOWN )
   END_RUNG
   RUNG wire#w1
      Contact( #IN_Empuj_Extendido )
      Coil( #EstadoVI.En_Empuj_Extendido )
   END_RUNG
   RUNG wire#w1
      Contact( #IN_Empuj_recogido )
      Coil( #EstadoVI.En_Empuj_Recogido )
   END_RUNG
   // the same network as SCL:
   #EstadoVI.En_Termico1 := true AND #Termico_Tx;
   #EstadoVI.En_PHS_1 := true AND #pHsMx_E1;
   #EstadoVI.En_PHS_3 := true AND #pHsMx_S3;
   #EstadoVI.En_Tope1_UP := true AND #TP1_Up AND NOT #TP1_Up;
   #EstadoVI.En_Tope1_DOWN := true AND NOT #TP1_Up AND #TP1_Down;
   #EstadoVI.En_Empuj_Extendido := true AND #IN_Empuj_Extendido;
   #EstadoVI.En_Empuj_Recogido := true AND #IN_Empuj_recogido;
END_REGION

REGION Network 56: Salidas Mesas
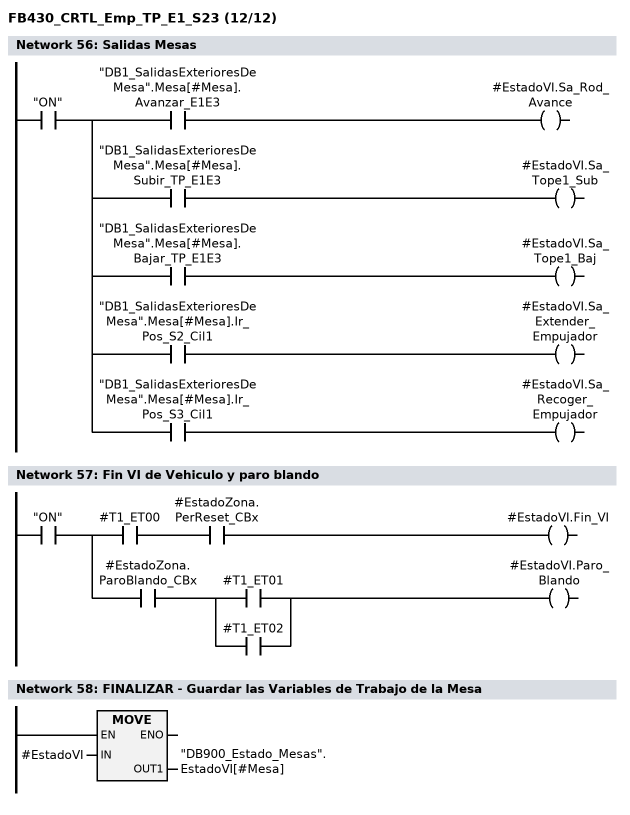
   RUNG wire#powerrail
      Contact( "ON" )
      wire#w1
      Contact( "DB1_SalidasExterioresDeMesa".Mesa[#Mesa].Avanzar_E1E3 )
      Coil( #EstadoVI.Sa_Rod_Avance )
   END_RUNG
   RUNG wire#w1
      Contact( "DB1_SalidasExterioresDeMesa".Mesa[#Mesa].Subir_TP_E1E3 )
      Coil( #EstadoVI.Sa_Tope1_Sub )
   END_RUNG
   RUNG wire#w1
      Contact( "DB1_SalidasExterioresDeMesa".Mesa[#Mesa].Bajar_TP_E1E3 )
      Coil( #EstadoVI.Sa_Tope1_Baj )
   END_RUNG
   RUNG wire#w1
      Contact( "DB1_SalidasExterioresDeMesa".Mesa[#Mesa].Ir_Pos_S2_Cil1 )
      Coil( #EstadoVI.Sa_Extender_Empujador )
   END_RUNG
   RUNG wire#w1
      Contact( "DB1_SalidasExterioresDeMesa".Mesa[#Mesa].Ir_Pos_S3_Cil1 )
      Coil( #EstadoVI.Sa_Recoger_Empujador )
   END_RUNG
   // the same network as SCL:
   #EstadoVI.Sa_Rod_Avance := "ON" AND "DB1_SalidasExterioresDeMesa".Mesa[#Mesa].Avanzar_E1E3;
   #EstadoVI.Sa_Tope1_Sub := "ON" AND "DB1_SalidasExterioresDeMesa".Mesa[#Mesa].Subir_TP_E1E3;
   #EstadoVI.Sa_Tope1_Baj := "ON" AND "DB1_SalidasExterioresDeMesa".Mesa[#Mesa].Bajar_TP_E1E3;
   #EstadoVI.Sa_Extender_Empujador := "ON" AND "DB1_SalidasExterioresDeMesa".Mesa[#Mesa].Ir_Pos_S2_Cil1;
   #EstadoVI.Sa_Recoger_Empujador := "ON" AND "DB1_SalidasExterioresDeMesa".Mesa[#Mesa].Ir_Pos_S3_Cil1;
END_REGION

REGION Network 57: Fin VI de Vehiculo y paro blando
   RUNG wire#powerrail
      Contact( "ON" )
      wire#w1
      Contact( #T1_ET00 )
      Contact( #EstadoZona.PerReset_CBx )
      Coil( #EstadoVI.Fin_VI )
   END_RUNG
   RUNG wire#w1
      Contact( #EstadoZona.ParoBlando_CBx )
      wire#w2
      Contact( #T1_ET01 )
      wire#w3
      Coil( #EstadoVI.Paro_Blando )
   END_RUNG
   RUNG wire#w2
      Contact( #T1_ET02 )
   END_RUNG wire#w3
   // the same network as SCL:
   #EstadoVI.Fin_VI := "ON" AND #T1_ET00 AND #EstadoZona.PerReset_CBx;
   #EstadoVI.Paro_Blando := "ON" AND #EstadoZona.ParoBlando_CBx AND (#T1_ET01 OR #T1_ET02);
END_REGION

REGION Network 58: FINALIZAR - Guardar las Variables de Trabajo de la Mesa
   RUNG wire#powerrail
      Move(in := #EstadoVI, out1 => "DB900_Estado_Mesas".EstadoVI[#Mesa])
   END_RUNG
   // the same network as SCL:
   "DB900_Estado_Mesas".EstadoVI[#Mesa] := #EstadoVI;
END_REGION
END_FUNCTION_BLOCK
